(* IEC 61131-3 sources: volt/packages/volt-lsp-iec/test-corpus/bakon-nano/Device/Plc Logic/Application/POUs/MachineControl, 14 files *)

(* ---- InputControl.pou ---- *)
PROGRAM InputControl
VAR
	bStartPressed		: BOOL;
	tonDelayStartButton : TON;
END_VAR
%LANGUAGE ST
(*TODO: IO Direct aan Station IO Hangen*)
//The quick brown fox jumps over the lazy dog

(*Data from IO *)
//Digital
g_byInputs_Module_00			:= %IB8;
g_byInputs_Module_01			:= %IB9;
//Analog
g_wInputs_Module_00				:= %IW5;
g_wInputs_Module_01				:= %IW6;

(*first  module *)
g_bDI_ES_DirectOK				:= g_byInputs_Module_00.0;
g_bDI_CircuitBreaker_i700		:= g_byInputs_Module_00.1;
g_bDI_CircuitBreaker_Ultrasonic	:= g_byInputs_Module_00.2;
g_bDI_PressureSwitchOK			:= g_byInputs_Module_00.3;
bStartPressed					:= g_byInputs_Module_00.4 OR (bStartPressed AND NOT tonDelayStartButton.q);
g_bDI_LightCurtainOK			:= g_byInputs_Module_00.5;
g_bDI_MachineInSafePosition		:= g_byInputs_Module_00.6;
g_bDI_TableCheck				:= g_byInputs_Module_00.7;

(*second module *)
g_bDI_Servo_Power_OK			:= g_byInputs_Module_01.0;
g_bDI_CleaningContainerUp		:= g_byInputs_Module_01.1;	//Spare
g_bDI_CleaningContainerDown		:= g_byInputs_Module_01.2;	//Spare
g_bDI_UltraSonic_Error			:= g_byInputs_Module_01.3;
g_bDI_UltraSonic_ErrorCode_1	:= g_byInputs_Module_01.4;
g_bDI_UltraSonic_ErrorCode_2	:= g_byInputs_Module_01.5;
g_bDI_Spare16					:= g_byInputs_Module_01.6;
g_bDI_Spare17					:= g_byInputs_Module_01.7;

tonDelayStartButton(IN:=bStartPressed, PT:=T#500MS);
g_bDI_StartButton := tonDelayStartButton.Q;

(*fifth module *)
g_iAI_UltrasonicPower			:= TO_INT(TO_REAL(g_wInputs_Module_00)/16384);
g_iAI_Spare_01					:= TO_INT(TO_REAL(g_wInputs_Module_01)/16384);

END_PROGRAM

(* ---- MACH_AUT_Automatic.pou ---- *)
PROGRAM MACH_AUT_Automatic
VAR
	tWatchDogTimer					: TON;
	tStepTimer						: TOF;
	bwait                  			: BOOL;
	bPulseStepCounter      			: BOOL;
	bHoldPointOnReq        			: BOOL;
	bHoldPointOnErr3       			: BOOL;
	bStopPointAutomatic    			: BOOL;

	bOnePiece						: BOOL;
	bStartButtonPressed				: BOOL;
	nOldProductType					: INT;
	nOldNumberRoundParts			: INT;
	nDebugLastStep					: INT;
	bStartedOnce						: BOOL := FALSE;
	rt_PressStartToInit: R_TRIG;
	tofRecipeLoad					: TOF;
	bStartPressedWhileLoadeing	: BOOL := FALSE;
	sOldRecipeName					: STRING;
	tMachineInSafePosition			: TOF;
	bFirstTimeWaitForExec: BOOL;
	nScanCount : INT;
	bStartPressedWhileError : BOOL;
END_VAR
%LANGUAGE ST
(*************************************************************************
 *
 * Application name			: Snijmachine
 * Module name				: MACH_AUT_automatic
 * Version number module	: 1.00
 *
 *
 *                  Copyright (c) Bakon 2009
 *                  Goes, The Netherlands
 *
 *
 * All rights are reserved. Reproduction in whole or in part is prohibited
 * without the written consent of the copyright owner.
 *
 *************************************************************************)

(*************************************************************************
 * HISTORY
 *************************************************************************
 * Update  :
 * Author  :
 * Changes :
 *************************************************************************)

(****************************************************************************************************************************)
bHoldPointOnReq		:= FALSE;
bHoldPointOnErr3		:= FALSE;
bStopPointAutomatic		:= FALSE;

g_sMACH.aut.bActAutomatic     := g_sMACH.MCL.bActAutomatic;

(* Force C_NOT_ACTIVE state *)
IF     NOT g_sMACH.aut.bActAutomatic
THEN
		IF g_sMACH.aut.nStepCounter <> C_NOT_ACTIVE THEN
			nDebugLastStep := g_sMACH.aut.nStepCounter;
		END_IF
		g_sMACH.aut.nStepCounter := C_NOT_ACTIVE;
END_IF;

IF         g_sMACH.aut.nStepCounter <> C_NOT_ACTIVE
THEN
   (* -------------------------------------------------------------------------
    * Prestep Code
    * ------------------------------------------------------------------------- *)
	tofRecipeLoad(IN:=g_HMI_sRecipeName <> sOldRecipeName, PT:=T#3s);
	sOldRecipeName := g_HMI_sRecipeName;
	bStartPressedWhileLoadeing := bStartPressedWhileLoadeing OR (tofRecipeLoad.Q AND g_bDI_StartButton);

	IF NOT gMachConfig.bCleaningUnit THEN		// Voor de veiligheid...
		g_bCleanRequest := FALSE;
	END_IF

END_IF

(* Product not finished reset when new recipe or when in Testmode *)
IF		g_HMI_RCP_Parameters.nProductType <> nOldProductType
	OR	g_HMI_RCP_Parameters.nPartsRound <> nOldNumberRoundParts
	OR	g_HMI_MachCommand.bTestMode
	OR 	g_HMI_MachCommand.bScanMode
	OR	g_sMACH.ERR.bCalcVerError
	OR	g_sMACH.ERR.bCalcHorError
	OR	g_sMACH.ERR.bCalcDia1Error
	OR	g_sMACH.ERR.bCalcDia2Error
	OR	g_sMACH.ERR.bErrorPosNotPossible
	OR	g_sMACH.ERR.bPieceTooLarge
	OR	g_sMACH.ERR.bTrayTooSmall
THEN
	g_bProductNotFinished := FALSE;
END_IF
nOldProductType := g_HMI_RCP_Parameters.nProductType;
nOldNumberRoundParts := g_HMI_RCP_Parameters.nPartsRound;

(* Offdelay g_bDI_MachineInSafePosition tbv veilig starten cyclus*)
tMachineInSafePosition(IN := g_bDI_MachineInSafePosition, PT := t#800ms);

(* detect change of state *)
bPulseStepCounter     := g_sMACH.aut.nStepCounter <> g_sMACH.aut.nOldStepCounter;
g_sMACH.aut.nOldStepCounter := g_sMACH.aut.nStepCounter;

(* Steptimer *)
tStepTimer (IN:=bPulseStepCounter, PT:= REAL_TO_TIME(g_sMACH.AUT.rStepTime));
bWait := tStepTimer.Q;

(* Watchdogtimer *)
tWatchdogTimer(	IN:=		NOT	bPulseStepCounter
							AND 		g_sMACH.AUT.bActAutomatic
							AND NOT 	g_sMACH.AUT.bAutomatichold
							AND NOT 	g_HMI_MachCommand.CMD.bResetErrorPulse
							AND 		g_sMACH.AUT.rWatchdogTime<> 0,
					PT:= 	REAL_TO_TIME(g_sMACH.AUT.rWatchdogTime));
g_sMACH.AUT.bAlmError := tWatchdogTimer.Q;

(* Melding op scherm om startknop in te drukken *)
rt_PressStartToInit(CLK := (g_sMACH.Aut.nStepCounter = C_INITIAL));
IF	rt_PressStartToInit.Q THEN
	g_sMACH.ERR.bPressStartToInit	:= TRUE;
END_IF
IF		g_bSUB_InitStart
	OR	(g_sMACH.Aut.nStepCounter = C_NOT_ACTIVE)
THEN
	g_sMACH.ERR.bPressStartToInit	:= FALSE;
END_IF
g_sMACH.ERR.bPressStartToCut	:= g_sMACH.Aut.nStepCounter = C_WAIT_EXEC;

CASE g_sMACH.Aut.nStepCounter OF
	(* --------------------------------------------------------------------------
	 * S-1  C_NOT_ACTIVE
	 *      OnEntry: Ready  := FALSE
	 *      OnEntry: Busy   := FALSE
	 *      OnEntry: Hold   := FALSE
	 *      OnEntry: Reset all non-stored commands
	 * T000 Activate signal
	 * -------------------------------------------------------------------------- *)
	C_NOT_ACTIVE:

		(* On Entry *)
		IF	bPulseStepCounter
		THEN
			g_sMACH.AUT.rWatchdogTime  			:= 0;
			g_sMACH.AUT.rStepTime				:= 0;

			g_sMACH.AUT.bAutomaticReady			:= FALSE;
			g_sMACH.AUT.bAutomaticBusy			:= FALSE;
			g_sMACH.AUT.bAutomaticHold			:= FALSE;
			g_sMACH.AUT.bAutomaticStop			:= FALSE;
			g_sMACH.AUT.bProcessBusy			:= FALSE;
			g_sMACH.AUT.bProcessReady			:= FALSE;
			g_sMACH.AUT.bAutomaticWaitingForTrig	:= FALSE;

			g_bCalculationStart					:= FALSE;
			g_bSUB_InitStart					:= FALSE;
			g_bSUB_CleanKnifeStart				:= FALSE;

			g_bCMD_US_Start1					:= FALSE;

			ModusRV.bEnable					:= FALSE;
			ModusRV.bStartXYA					:= FALSE;
			ModusRV.bStartZ						:= FALSE;

			g_sHMI_Mach_UnitStatus.bProcessAgain	:= FALSE;
			bStartButtonPressed							:= FALSE;

			g_bSaveMachPar								:= bStartedOnce;

			g_HMI_MachCommand.CMD.bDeny			:= FALSE;
			g_HMI_MachCommand.CMD.bConfirm		:= FALSE;

			bStartPressedWhileLoadeing := FALSE;
			g_sMACH.ERR.bMessagePosNotPossible := FALSE;

			g_HMI_MachCommand.CMD.bCleanKnifeRequest	:= FALSE;
			g_sHMI_Mach_UnitStatus.bPopupRemoveProduct := FALSE;
		END_IF

		(* Continuous actions *)
		IF NOT g_HMI_MachCommand.bScanMode THEN
			nScanCount := 0;
		END_IF

		(* Transitions *)
		IF	g_sMACH.aut.bActAutomatic
		THEN
			g_sMACH.aut.nStepCounter         := C_INITIAL;
			bStartedOnce := TRUE;
		END_IF;

	(* --------------------------------------------------------------------------
	 * S000 Sub init before starting auto cycle
	 * T995 C_WAIT_EXEC, Pre init done
	 * -------------------------------------------------------------------------- *)
	C_INITIAL:

	      (* On Entry *)
	      IF	bPulseStepCounter
		THEN
			g_sMACH.AUT.rWatchdogTime  			:= 0;
			g_sMACH.AUT.rStepTime				:= 0;
			MACH_SUB_Initialise.I_rX_InfeedPosition		:= g_HMI_MCH_Parameters.rInfeedPosition_X;
			IF 		g_HMI_MachCommand.bTestMode
				OR 	g_HMI_MachCommand.bScanMode
			THEN
				MACH_SUB_Initialise.I_rY_InfeedPosition		:= g_HMI_MCH_Parameters.rInfeedPosition_Y + 30;
			ELSE
				MACH_SUB_Initialise.I_rY_InfeedPosition		:= g_HMI_MCH_Parameters.rInfeedPosition_Y;
			END_IF
			MACH_SUB_Initialise.I_rY_InfeedPrePosition	:= g_HMI_MCH_Parameters.rInfeedPosition_Y + 30;
		END_IF;

		(* Continuous actions *)
		IF	g_bDI_StartButton OR g_HMI_MachCommand.bScanMode
		THEN
			g_bSUB_InitStart							:= TRUE;
		END_IF

		(* Transitions *)
		IF		g_bSUB_InitDone
		THEN
				g_bSUB_InitStart				:= FALSE;
				g_sMACH.aut.nStepCounter	:= C_WAIT_EXEC;
				bStartPressedWhileLoadeing := FALSE;
		END_IF;

	(* --------------------------------------------------------------------------
	 * S995 C_WAIT_EXEC
	 *      AutomaticWaitingForTrig := NOT AutomaticStop
	 * T996 C_INITIALISE
	 *              Execution Trigger
	 *      AND NOT Hold On Request
	 *      AND NOT Hold On Error Category 3
	 *      AND NOT Stop end of cycle selected
	 *      AND NOT Stop at error category 2
	 * T997 C_STOPPED
	 *         "Stop end of cycle" selected
	 *      OR "Stop on error category 2"
	 * -------------------------------------------------------------------------- *)
	C_WAIT_EXEC:

	      (* Actions on state entry *)
		IF	bPulseStepCounter
		THEN
			g_sMACH.AUT.rWatchdogTime  			:= 0;
			g_sMACH.AUT.rStepTime				:= 0;
			g_sMACH.ERR.bMessagePosNotPossible := FALSE;
			g_sMACH.AUT.rWatchdogTime  			:= 0;
			IF	g_HMI_MachCommand.bScanMode AND NOT bFirstTimeWaitForExec THEN
				g_sMACH.AUT.rStepTime			:= 2000;
			ELSE
				g_sMACH.AUT.rStepTime				:= 0;
			END_IF
			IF g_sMACH.ERR.bCrashDetected THEN
				g_bProductNotFinished	:= FALSE;
				g_sHMI_Mach_UnitStatus.bPopupRemoveProduct	:= TRUE;	// Popup
			END_IF
			bStartPressedWhileError := FALSE;
		END_IF

		bStartPressedWhileError := bStartPressedWhileError OR (g_sMACH.ERR.bCrashDetected AND g_bDI_StartButton);

		(* Continuous actions *)
		bHoldPointOnReq     := TRUE;
		bHoldPointOnErr3    := TRUE;
		bStopPointAutomatic := TRUE;
		IF	g_HMI_MachCommand.CMD.bConfirm THEN
			g_sHMI_Mach_UnitStatus.bPopupRemoveProduct	:= FALSE;	// Popup
			g_HMI_MachCommand.CMD.bConfirm	:= FALSE;
			g_sMACH.ERR.bCrashDetected	:= FALSE;
		END_IF

		(* Transitions *)
		IF				g_sMACH.MCL.bStopEndOfCycle
				OR		g_sMACH.MCL.bStopOnErrorCat2
				OR 		(g_HMI_MachCommand.bScanMode AND nScanCount >= 10)
		THEN
			g_sMACH.aut.nStepCounter     		:= C_STOPPED;
			IF g_HMI_MachCommand.bScanMode THEN
				g_sHMI_Mach_UnitStatus.bScanFinished := TRUE;
				g_bScanDataPending := TRUE;
			END_IF
		ELSIF	((g_bDI_StartButton
			AND tMachineInSafePosition.Q)
			OR g_HMI_MachCommand.bTestMode
			OR	(g_HMI_MachCommand.bScanMode
			AND NOT bwait AND nScanCount < 10)
			OR (bStartPressedWhileLoadeing
			AND tMachineInSafePosition.Q)
			OR bStartPressedWhileError)
			AND g_bDI_LightCurtainOK
			AND NOT tofRecipeLoad.Q
			AND NOT g_sMACH.ERR.bCrashDetected
		THEN
			g_uControl_X_Axis.bEnableDrive		:= TRUE;
			g_uControl_Y_Axis.bEnableDrive		:= TRUE;
			g_uControl_Front_Axis.bEnableDrive	:= TRUE;
			g_uControl_Rear_Axis.bEnableDrive	:= TRUE;
			g_uControl_Z_Axis.bEnableDrive		:= TRUE;
			g_uControl_R_Axis.bEnableDrive		:= TRUE;

			bStartButtonPressed 				:= FALSE;
			bStartPressedWhileLoadeing	:= FALSE;
			g_sMACH.aut.nStepCounter		:= C_INITIALISE;
		END_IF

	(* --------------------------------------------------------------------------
	 * S996 C_INITIALISE
	 *      OnEntry: bProcessBusy  := TRUE
	 *      OnEntry: ProcessReady := FALSE
	 * T005 Always
	 * -------------------------------------------------------------------------- *)
	C_INITIALISE:

	      (* On entry *)
		IF	bPulseStepCounter
		THEN
			g_sMACH.aut.bProcessReady		:= FALSE;
			g_sMACH.aut.bProcessBusy		:= TRUE;
			g_sMACH.AUT.rWatchdogTime  		:= 10 * 1000;
			g_sMACH.AUT.rStepTime			:= 0;
	      END_IF

		(* Continuous actions *)
		IF g_sMACH.AUT.bAlmError THEN
			IF NOT g_uStatus_X_Axis.bDriveEnabled
				OR NOT g_uStatus_Y_Axis.bDriveEnabled
				OR NOT g_uStatus_Front_Axis.bDriveEnabled
				OR NOT g_uStatus_Rear_Axis.bDriveEnabled
			THEN
				g_sMACH.ERR.bXYNotEnabled := TRUE;
			END_IF
			IF NOT g_uStatus_Z_Axis.bDriveEnabled THEN
				g_sMACH.ERR.bZNotEnabled := TRUE;
			END_IF
			IF NOT g_uStatus_R_Axis.bDriveEnabled THEN
				g_sMACH.ERR.bRNotEnabled := TRUE;
			END_IF
		END_IF
		IF	g_HMI_MachCommand.CMD.bConfirm THEN
			g_sHMI_Mach_UnitStatus.bPopupRemoveProduct	:= FALSE;	// Popup
			g_HMI_MachCommand.CMD.bConfirm	:= FALSE;
			g_sMACH.ERR.bCrashDetected	:= FALSE;
		END_IF

		(* Transitions *)
		IF		g_uStatus_Z_Axis.bDriveEnabled
			AND	g_uStatus_R_Axis.bDriveEnabled
			AND	g_uStatus_X_Axis.bDriveEnabled
			AND	g_uStatus_Y_Axis.bDriveEnabled
			AND	g_uStatus_Rear_Axis.bDriveEnabled
			AND	g_uStatus_Front_Axis.bDriveEnabled
			AND NOT g_sMACH.ERR.bCrashDetected
		THEN
			g_sMACH.aut.nStepCounter	:= 010;
		END_IF

	(*--------------------------------------------------------------------------
	 * S010 Enable Modus RondVierkant
	 *		 Check if product has been cut completely
	 * T015 Always
	 * -------------------------------------------------------------------------- *)
	010:

	      (* On entry *)
		IF	bPulseStepCounter
		THEN
			g_sMACH.AUT.rWatchdogTime  				:= 0;
			g_sMACH.AUT.rStepTime					:= 0;
			ModusRV.bEnable 							:= TRUE;
			IF g_bProductNotFinished AND NOT g_HMI_MachCommand.bTestMode AND NOT g_HMI_MachCommand.bScanMode
			THEN
				g_sHMI_Mach_UnitStatus.bProcessAgain	:= TRUE;	(* Open popup in screen *)
			END_IF
		END_IF

		(* Continuous actions *)

		(* Transitions *)
		IF			(g_bProductNotFinished AND g_HMI_MachCommand.CMD.bDeny)
			OR		g_HMI_MachCommand.bTestMode
			OR 		g_HMI_MachCommand.bScanMode
			OR	NOT	g_bProductNotFinished
		THEN
			g_sHMI_Mach_UnitStatus.bProcessAgain	:= FALSE;	(* Popup in screen *)
			g_HMI_MachCommand.CMD.bDeny			:= FALSE;
			g_HMI_MachCommand.CMD.bConfirm		:= FALSE;
			g_sMACH.aut.nStepCounter	:= 015;
		ELSIF	(g_bProductNotFinished AND g_HMI_MachCommand.CMD.bConfirm)
		THEN
			g_sHMI_Mach_UnitStatus.bProcessAgain	:= FALSE;	(* Popup in screen *)
			g_HMI_MachCommand.CMD.bDeny			:= FALSE;
			g_HMI_MachCommand.CMD.bConfirm		:= FALSE;
			g_sMACH.aut.nStepCounter	:= 020;
		END_IF

	(*--------------------------------------------------------------------------
	 * S015 Calculate cutting positions
	 * T020 Calculations done
	 * -------------------------------------------------------------------------- *)
	015:

	      (* On entry *)
		IF	bPulseStepCounter
		THEN
			g_sMACH.AUT.rWatchdogTime  				:= 0;
			g_sMACH.AUT.rStepTime					:= 0;
			g_bCalculationStart							:= TRUE;

		END_IF

		(* Continuous actions *)
		bOnePiece	:= 		g_HMI_RCP_Parameters.rSizeTrimRight = 0 												(* No cuts when one piece and no trims *)
					AND	g_HMI_RCP_Parameters.rSizeTrimLeft = 0
					AND	g_HMI_RCP_Parameters.rSizeTrimRear = 0
					AND	g_HMI_RCP_Parameters.rSizeTrimFront = 0
					AND	g_HMI_RCP_Parameters.nPartsX = 1
					AND	g_HMI_RCP_Parameters.nPartsY = 1;

		(* Transitions *)
		IF			g_bCalculationDone
		THEN
			g_bCalculationStart				:= FALSE;
			g_sMACH.aut.nStepCounter		:= 020;
		END_IF

	(*--------------------------------------------------------------------------
	 * S020 Start cutting
	 * T025 Always
	 * -------------------------------------------------------------------------- *)
	020:

	      (* On entry *)
		IF	bPulseStepCounter
		THEN
			g_sMACH.AUT.rWatchdogTime  				:= 0;
			g_sMACH.AUT.rStepTime					:= 0;
			IF	NOT bOnePiece
			THEN
				ModusRV.bStartXYA	:= TRUE;
				ModusRV.bStartZ		:= TRUE;
				g_bProductNotFinished	:= TRUE;
				g_bCMD_US_Start1	:= TRUE;
			END_IF
		END_IF

		(* Continuous actions *)

		(* Transitions *)
		IF	TRUE
		THEN
			g_sMACH.aut.nStepCounter	:= 025;
		END_IF

	(*--------------------------------------------------------------------------
	 * S025 Wait for cutting ready
	 * T030 Cutting ready
	 * -------------------------------------------------------------------------- *)
	025:

	    (* On entry *)
		IF	bPulseStepCounter
		THEN
			g_sMACH.AUT.rWatchdogTime  				:= 0;
			g_sMACH.AUT.rStepTime					:= 0;
		END_IF

		(* Continuous actions *)

		(* Transitions *)
		IF		ModusRV.bLastCutReadyZOutOfProduct
			OR	ModusRV.bReady									(* @TODO, tekst bijzetten waarom, vermoedelijk voor als een product geen enkele keer gesneden moet worden *)
		THEN
			ModusRV.bStartXYA		:= FALSE;
			ModusRV.bStartZ			:= FALSE;
			g_bProductNotFinished	:= FALSE;
			g_sHMI_CountersInfinite.dnProductCountTotal	:= g_sHMI_CountersInfinite.dnProductCountTotal + 1;
			g_sHMI_CountersDay.dnProductCountTotal	:= g_sHMI_CountersDay.dnProductCountTotal + 1;
			g_bCMD_US_Start1	:= FALSE;

			IF NOT g_HMI_MachCommand.bScanMode AND NOT g_sMACH.ERR.bCrashDetected THEN
				CASE g_HMI_RCP_Parameters.nProductType OF
						Prod_Slab_Rectangle_1x1, Prod_Slab_Rectangle_1x1_Clamp:	(* ProductType = 0 = Slab Square *)
							g_sHMI_CountersInfinite.dnProductCountSlabSquare	:= 	g_sHMI_CountersInfinite.dnProductCountSlabSquare	+1;
							g_sHMI_CountersDay.dnProductCountSlabSquare		:= 	g_sHMI_CountersDay.dnProductCountSlabSquare	+1;
						Prod_Slab_Triangle_1x1:	(* ProductType = 1 = Slab triangle *)
							g_sHMI_CountersInfinite.dnProductCountSlabTriangle	:= 	g_sHMI_CountersInfinite.dnProductCountSlabTriangle	+1;
							g_sHMI_CountersDay.dnProductCountSlabTriangle	:= 	g_sHMI_CountersDay.dnProductCountSlabTriangle	+1;
						Prod_Slab_Diagonal_1x1:	(* ProductType = 2 = Slab diagonal *)
							g_sHMI_CountersInfinite.dnProductCountSlabDiagonal	:= 	g_sHMI_CountersInfinite.dnProductCountSlabDiagonal	+1;
							g_sHMI_CountersDay.dnProductCountSlabDiagonal		:= 	g_sHMI_CountersDay.dnProductCountSlabDiagonal	+1;
						Prod_Round_POC_2x1:	(* ProductType = 4 = Round Cake *)
							g_sHMI_CountersInfinite.dnProductCountRound		:= 	g_sHMI_CountersInfinite.dnProductCountRound + 2;
							g_sHMI_CountersDay.dnProductCountRound			:= 	g_sHMI_CountersDay.dnProductCountRound + 2;
						Prod_Tray_Rectangle_1x2, Prod_Tray_Rectangle_2x1:	(* ProductType = 4 = Tray Square Small *)
							g_sHMI_CountersInfinite.dnProductCountTraySmall		:= 	g_sHMI_CountersInfinite.dnProductCountTraySmall + 2;
							g_sHMI_CountersDay.dnProductCountTraySmall			:= 	g_sHMI_CountersDay.dnProductCountTraySmall + 2;
						Prod_Tray_Rectangle_1x1:	(* ProductType = 5 = Tray Square Large *)
							g_sHMI_CountersInfinite.dnProductCountTrayLarge		:= 	g_sHMI_CountersInfinite.dnProductCountTrayLarge +1;
							g_sHMI_CountersDay.dnProductCountTrayLarge			:= 	g_sHMI_CountersDay.dnProductCountTrayLarge +1;
						Prod_Tray_Rectangle_1x4:	(* ProductType =6 = Tray Square Triple *)
							g_sHMI_CountersInfinite.dnProductCountTrayTriple		:= 	g_sHMI_CountersInfinite.dnProductCountTrayTriple + 4;
							g_sHMI_CountersDay.dnProductCountTrayTriple			:= 	g_sHMI_CountersDay.dnProductCountTrayTriple + 4;
				END_CASE
			END_IF
			g_sMACH.aut.nStepCounter	:= 030;
		ELSIF	bOnepiece
		THEN
			ModusRV.bStartXYA			:= FALSE;
			ModusRV.bStartZ				:= FALSE;
			g_bProductNotFinished		:= FALSE;
			g_bCMD_US_Start1			:= FALSE;
			g_sMACH.aut.nStepCounter	:= 030;
		END_IF

	(*--------------------------------------------------------------------------
	 * S030 Wait for Modus ready
	 * T040 Cleaning
	 * T998 Modus ready
	 * -------------------------------------------------------------------------- *)
	030:

	      (* On entry *)
		IF	bPulseStepCounter
		THEN
			g_sMACH.AUT.rWatchdogTime  				:= 0;
			g_sMACH.AUT.rStepTime					:= 0;
		END_IF

		(* Continuous actions *)

		(* Transitions *)
		IF			ModusRV.bReady
				OR	bOnePiece
		THEN
(*			g_uControl_Front_Axis.bEnableDrive	:= FALSE;
			g_uControl_Rear_Axis.bEnableDrive	:= FALSE;
			g_uControl_Z_Axis.bEnableDrive		:= FALSE;
			g_uControl_R_Axis.bEnableDrive		:= FALSE;*)
			(*IF	g_bCleanRequest
			THEN
				g_bCleanRequest	:= FALSE;
				g_HMI_MachCommand.CMD.bCleanKnifeRequest	:= FALSE;
				g_sMACH.aut.nStepCounter	:= 40;
			ELSE *)
			g_uControl_X_Axis.bEnableDrive := FALSE;
			g_uControl_Y_Axis.bEnableDrive := FALSE;
			//g_HMI_MachCommand.CMD.bCleanKnifeRequest	:= FALSE;
			nScanCount := nScanCount + 1;
			g_sMACH.aut.nStepCounter	:= C_READY;
			//END_IF
		END_IF

	(*--------------------------------------------------------------------------
	 * S040 Cleaning
	 * T998 Modus ready
	 * -------------------------------------------------------------------------- *)
	040:

	      (* On entry *)
		IF	bPulseStepCounter
		THEN
			g_sMACH.AUT.rWatchdogTime  			:= 0;
			g_sMACH.AUT.rStepTime				:= 0;
			g_bSUB_CleanKnifeStart				:= TRUE;
		END_IF

		(* Continuous actions *)

		(* Transitions *)
		IF	g_bSUB_CleanKnifeDone
		THEN
(*			g_uControl_Front_Axis.bEnableDrive	:= FALSE;
			g_uControl_Rear_Axis.bEnableDrive	:= FALSE;
			g_uControl_Z_Axis.bEnableDrive		:= FALSE;
			g_uControl_R_Axis.bEnableDrive		:= FALSE;*)
			g_uControl_X_Axis.bEnableDrive	:= FALSE;
			g_uControl_Y_Axis.bEnableDrive	:= FALSE;
			g_bSUB_CleanKnifeStart			:= FALSE;
			g_sMACH.aut.nStepCounter		:= C_READY;
		END_IF

	(* --------------------------------------------------------------------------
	 * S998 C_READY
	 *      OnEntry: bProcessBusy  := FALSE
	 *      OnEntry: ProcessReady := TRUE
	 * T999 Always
	 * -------------------------------------------------------------------------- *)
	C_READY:

	      (* On Entry *)
		IF	bPulseStepCounter
		THEN
			g_sMACH.aut.bProcessBusy		:= FALSE;
			g_sMACH.aut.bProcessReady	:= TRUE;
			g_sMACH.aut.rWatchdogTime	:= 0;
		END_IF

		(* Continuous actions *)

		(* Transitions *)
		IF	TRUE
		THEN
			g_sMACH.AUT.rStepTime	:= 0;
			g_sMACH.aut.nStepCounter	:= C_LAST;
		END_IF

	(* --------------------------------------------------------------------------
	 * S997 C_STOPPED
	 *      OnEntry: AutomaticReady := TRUE
	 * T999     NOT "Stop end of cycle" selected
	 *      AND NOT "Stop on error category 2"
	 * -------------------------------------------------------------------------- *)
	C_STOPPED:

		(* On entry *)
		IF	bPulseStepCounter
		THEN
			g_sMACH.aut.rWatchdogTime     := 0;
		END_IF

		(* Continuous actions *)
		(*g_uControl_X_Axis.bEnableDrive	:=	FALSE; //g_uStatus_X_Axis.bAutomaticEnabled;
		g_uControl_Y_Axis.bEnableDrive	:=	FALSE; //g_uStatus_Y_Axis.bAutomaticEnabled;
		g_uControl_Front_Axis.bEnableDrive := FALSE; //g_uStatus_Front_Axis.bAutomaticEnabled;
		g_uControl_Rear_Axis.bEnableDrive := FALSE; //g_uStatus_Rear_Axis.bAutomaticEnabled;
		g_uControl_Z_Axis.bEnableDrive	:=	FALSE; //g_uStatus_Z_Axis.bAutomaticEnabled;
		g_uControl_R_Axis.bEnableDrive	:=	FALSE; //g_uStatus_R_Axis.bAutomaticEnabled;*)
		bStopPointAutomatic				:= TRUE;

		g_sMACH.Aut.bAutomaticReady    := TRUE;(*NOT (
													g_uStatus_X_Axis.bDriveEnabled
												OR	g_uStatus_Y_Axis.bDriveEnabled
												OR	g_uStatus_Front_Axis.bDriveEnabled
												OR	g_uStatus_Rear_Axis.bDriveEnabled
												OR	g_uStatus_Z_Axis.bDriveEnabled);*)

		(* Transitions *)
		IF		NOT g_sMACH.MCL.bStopEndOfCycle
			AND NOT g_sMACH.MCL.bStopOnErrorCat2
			AND NOT g_sHMI_Mach_UnitStatus.bScanFinished
		THEN
			g_sMACH.Aut.bAutomaticReady   := FALSE;
			g_sMACH.aut.nStepCounter      := C_LAST;
		END_IF

	(* --------------------------------------------------------------------------
	 * S999 C_LAST
	 * T000 Always
	 * -------------------------------------------------------------------------- *)
	C_LAST:

		(* On entry *)
		IF	bPulseStepCounter
		THEN
			g_sMACH.aut.rWatchdogTime     := 0;
		END_IF

		(* Continuous actions *)

		(* Transitions *)
		IF	TRUE THEN
			g_sMACH.aut.nStepCounter      := C_WAIT_EXEC;
		END_IF

	(* --------------------------------------------------------------------------
	 * Illegal state
	 * -------------------------------------------------------------------------- *)
ELSE
	g_sMACH.aut.rWatchdogTime     := 10;
END_CASE

IF      g_sMACH.Aut.nStepCounter <> C_NOT_ACTIVE
THEN
	(* --------------------------------------------------------------------------
	 * Poststep code
	 * -------------------------------------------------------------------------- *)
	g_sMACH.Aut.bAutomaticHold  :=	(	g_sMACH.MCL.bHoldOnRequest
									AND	bHoldPointOnReq)
									OR  (    g_sMACH.MCL.bHoldOnErrorCat3
									AND bHoldPointOnErr3);

	g_sMACH.Aut.bAutomaticStop  :=			bStopPointAutomatic
									AND	g_sMACH.MCL.bStopOnErrorCat2;

	g_sMACH.Aut.bAutomaticBusy  :=		NOT	g_sMACH.Aut.bAutomaticHold
										AND NOT	g_sMACH.Aut.bAutomaticStop;

	g_sMACH.Aut.bAutomaticWaitingForTrig :=        (g_sMACH.aut.nStepCounter = C_WAIT_EXEC)
												AND NOT g_sMACH.Aut.bAutomaticStop
												AND NOT g_sMACH.Aut.bAutomaticHold;
	g_sHMI_Mach_UnitStatus.nScanProgress := nScanCount;
END_IF

END_PROGRAM

(* ---- MACH_Call.pou ---- *)
PROGRAM MACH_Call
VAR
END_VAR
%LANGUAGE ST
(*************************************************************************
 *
 * Application name			: Snijmachine
 * Module name				: MACH_Call
 * Version number module	: 0.00
 *
 *                  Copyright (c) Bakon 2009
 *                  Goes, The Netherlands
 *
 *
 * All rights are reserved. Reproduction in whole or in part is prohibited
 * without the written consent of the copyright owner.
 *
 *************************************************************************)

(*************************************************************************
 * HISTORY
 *************************************************************************
 * Update  :
 * Author  :
 * Changes :
 *************************************************************************)

	(* -------------------------------------------------------------------------
	* Execution Control functions
	* ------------------------------------------------------------------------- *)
	MACH_HMI_Control();

	(* -------------------------------------------------------------------------
	* Execution Control functions
	* ------------------------------------------------------------------------- *)
	MACH_INI_Initialise();
(*    MACH_AUT_Automatic(); *)
	MACH_MAN_Manual();
	MACH_ERH_ErrorHandler();
	MACH_MCL_ModeControl();
	MACH_CLN_Cleaning();

	(* -------------------------------------------------------------------------
	* Drivers and calculations
	* ------------------------------------------------------------------------- *)
	MACH_DRV_DriverCall();
	Calc_Main();	(* Calculations *)

	(* -------------------------------------------------------------------------
	* Miscellaneous
	* ------------------------------------------------------------------------- *)
	MACH_MIS_Miscellaneous();
	MACH_ParameterHandler();
	RCP_RecipeHandler();
	HMI_ResetSignals();
	{warning 'Disabled for compatibility - SVE'}
	//g_Logger(directoryName := '/USBStorage/IPC/PLC/KC_Logs');

END_PROGRAM

(* ---- MACH_CLN_Cleaning.pou ---- *)
PROGRAM MACH_CLN_Cleaning
VAR
	bPulseStepCounter	: BOOL;
	bWait				: BOOL;
	tWatchDogTimer		: TON;
	tStepTimer			: TOF;
	rt_PressStartToInit	: R_TRIG;
END_VAR
%LANGUAGE ST
 (*************************************************************************
 *
 * Application name				: Snijmachine
 * Module name					: MACH_CLN_Cleaning
 * Version number module		: 0.00
 *
 *
 *						Copyright (c) Bakon 2009
 *						Goes, The Netherlands
 *
 *
 * All rights are reserved. Reproduction in whole or in part is prohibited
 * without the written consent of the copyright owner.
 *
 *************************************************************************)

(*************************************************************************
 * HISTORY
 *************************************************************************
 * Update  :
 * Author  :
 * Changes :
 *************************************************************************)

(* Force C_NOT_ACTIVE state *)
IF	NOT g_sMACH.MCL.bActCleaning
THEN
	g_sMACH.CLN.nStepCounter := C_NOT_ACTIVE;
END_IF;

IF		g_sMACH.CLN.nStepCounter <> C_NOT_ACTIVE
THEN
	(* -------------------------------------------------------------------------
	 * Prestep Code
	 * ------------------------------------------------------------------------- *)
				  ;
END_IF;

(* detect change of state *)
bPulseStepCounter	  := g_sMACH.CLN.nStepCounter <> g_sMACH.CLN.nOldStepCounter;
g_sMACH.CLN.nOldStepCounter := g_sMACH.CLN.nStepCounter;

(* Steptimer *)
tStepTimer (IN:= bPulseStepCounter, PT:= REAL_TO_TIME(g_sMACH.CLN.rStepTime));
bWait := tStepTimer.Q;

(* Watchdogtimer *)
tWatchDogTimer (IN:= 	NOT	bPulseStepCounter
					AND		g_sMACH.MCL.bActCleaning
					AND NOT	g_HMI_MachCommand.CMD.bResetErrorPulse
					AND		g_sMACH.CLN.rWatchdogTime <> 0,
				PT:= REAL_TO_TIME(g_sMACH.CLN.rWatchdogTime));
g_sMACH.CLN.bAlmError := tWatchDogTimer.Q;

(* Melding op scherm om startknop in te drukken *)
rt_PressStartToInit(CLK := (g_sMACH.CLN.nStepCounter = C_INITIAL));
IF	rt_PressStartToInit.Q THEN
	g_sMACH.ERR.bPressStartToCleanInit	:= TRUE;
END_IF
IF		g_bSUB_InitStart
	OR	(g_sMACH.CLN.nStepCounter = C_NOT_ACTIVE)
THEN
	g_sMACH.ERR.bPressStartToCleanInit	:= FALSE;
END_IF

CASE g_sMACH.CLN.nStepCounter OF
	(* --------------------------------------------------------------------------
	 * S-1  C_NOT_ACTIVE
	 *		OnEntry: Ready  := FALSE
	 *		OnEntry: Busy	:= FALSE
	 *		OnEntry: Reset all non-stored commands
	 * T000 Activate signal
	 * -------------------------------------------------------------------------- *)
	C_NOT_ACTIVE:

		(* On Entry *)
		IF		bPulseStepCounter
		THEN
				g_sMACH.CLN.rWatchdogTime					:= 0;
				g_sMACH.CLN.bCleaningReady					:= FALSE;
				g_sMACH.CLN.bCleaningBusy					:= FALSE;

				g_bSUB_InitStart							:= FALSE;

				g_HMI_MachCommand.CMD.bCleanKnifeRequest		:= FALSE;
				g_bSUB_CleanKnifeStart							:= FALSE;
				g_sHMI_Mach_UnitStatus.bKnifeCleaningBusy		:= FALSE;

				g_bCMD_US_Start1 							:= FALSE;
		END_IF

		(* Continuous actions *)

		(* Transitions *)
		IF		g_sMACH.MCL.bActCleaning
		THEN
				g_sMACH.CLN.nStepCounter			:= C_INITIAL;
		END_IF

	(* --------------------------------------------------------------------------
	 * S000 C_INITIAL
	 *		OnEntry: Ready := FALSE
	 *		OnEntry: Busy  := TRUE
	 *		Enable drives
	 * T001 Drives enabled
	 * -------------------------------------------------------------------------- *)
	C_INITIAL:

		(* On Entry *)
		IF		bPulseStepCounter
		THEN
				g_sMACH.CLN.rWatchdogTime					:= 0;
				g_sMACH.CLN.bCleaningReady					:= FALSE;
				g_sMACH.CLN.bCleaningBusy					:= TRUE;
		END_IF

		(* Continuous actions *)

		(* Transitions *)
		IF		g_sMACH.MCL.bStopEndOfCycle
		THEN
				g_sMACH.CLN.nStepCounter			:= C_READY;
		ELSIF			g_bDI_StartButton
				OR NOT	g_bDI_MachineInSafePosition
		THEN
				g_sMACH.CLN.nStepCounter			:= 005;
		END_IF

	(* --------------------------------------------------------------------------
	 * S005 Sub init before starting cleaning
	 * T010 Cleaning
	 * -------------------------------------------------------------------------- *)

	005:
		(* On Entry *)
	    IF	bPulseStepCounter
		THEN
			g_sMACH.CLN.rWatchdogTime  			:= 0;
			g_sMACH.CLN.rStepTime				:= 0;
			MACH_SUB_Initialise.I_rX_InfeedPosition		:= g_HMI_MCH_Parameters.rInfeedPosition_X;
			MACH_SUB_Initialise.I_rY_InfeedPosition		:= g_HMI_MCH_Parameters.rInfeedPosition_Y + 30;
			MACH_SUB_Initialise.I_rY_InfeedPrePosition	:= g_HMI_MCH_Parameters.rInfeedPosition_Y + 30;
		END_IF

		g_bSUB_InitStart						:= TRUE;

		(* Transitions *)
		IF	g_bSUB_InitDone
		THEN
			g_sMACH.CLN.nStepCounter			:= 010;
			g_bSUB_InitStart := FALSE;
		END_IF

	(* --------------------------------------------------------------------------
	 * S010 Enable drives
	 * T015 Drives enabled
	 * -------------------------------------------------------------------------- *)
	010:

		(* On Entry *)
		IF		 bPulseStepCounter
		THEN
				g_sMACH.CLN.rWatchdogTime			:= 10*1000;
				g_sMACH.CLN.rStepTime				:= 0;
				g_uControl_X_Axis.bEnableDrive		:= TRUE;
				g_uControl_Y_Axis.bEnableDrive		:= TRUE;
				g_uControl_Front_Axis.bEnableDrive	:= TRUE;
				g_uControl_Rear_Axis.bEnableDrive	:= TRUE;
				g_uControl_Z_Axis.bEnableDrive		:= TRUE;
				g_uControl_R_Axis.bEnableDrive		:= TRUE;
		END_IF

		(* Continuous actions *)
		IF g_sMACH.CLN.bAlmError THEN
			IF NOT g_uStatus_X_Axis.bDriveEnabled
				OR NOT g_uStatus_Y_Axis.bDriveEnabled
				OR NOT g_uStatus_Front_Axis.bDriveEnabled
				OR NOT g_uStatus_Rear_Axis.bDriveEnabled
			THEN
				g_sMACH.ERR.bXYNotEnabled := TRUE;
			END_IF
			IF NOT g_uStatus_Z_Axis.bDriveEnabled THEN
				g_sMACH.ERR.bZNotEnabled := TRUE;
			END_IF
			IF NOT g_uStatus_R_Axis.bDriveEnabled THEN
				g_sMACH.ERR.bRNotEnabled := TRUE;
			END_IF
		END_IF

		(* Transitions *)
		IF		g_uStatus_Z_Axis.bDriveEnabled// AND g_uStatus_Z_Axis.bAutomaticEnabled
			AND	g_uStatus_R_Axis.bDriveEnabled //AND g_uStatus_R_Axis.bAutomaticEnabled
			AND	g_uStatus_X_Axis.bDriveEnabled //AND g_uStatus_X_Axis.bAutomaticEnabled
			AND	g_uStatus_Y_Axis.bDriveEnabled //AND g_uStatus_Y_Axis.bAutomaticEnabled
			AND	g_uStatus_Rear_Axis.bDriveEnabled //AND g_uStatus_Rear_Axis.bAutomaticEnabled
			AND	g_uStatus_Front_Axis.bDriveEnabled //AND g_uStatus_Front_Axis.bAutomaticEnabled
		THEN
				  g_sMACH.CLN.nStepCounter				:= 15;
		END_IF

	(* --------------------------------------------------------------------------
	 * S015 Wait for request from HMI
	 * T020	Start cleaning
	 * T998 Never
	 * -------------------------------------------------------------------------- *)
	015:

		(* On Entry *)
		IF		 bPulseStepCounter
		THEN
				g_sMACH.CLN.rWatchdogTime			:= 0;
				g_sMACH.CLN.rStepTime				:= 0;
				//g_uControl_X_Axis.bEnableDrive		:= TRUE;
				//g_uControl_Y_Axis.bEnableDrive		:= TRUE;
				//g_uControl_Front_Axis.bEnableDrive	:= TRUE;
				//g_uControl_Rear_Axis.bEnableDrive	:= TRUE;
				//g_uControl_Z_Axis.bEnableDrive		:= TRUE;
				//g_uControl_R_Axis.bEnableDrive		:= TRUE;
				g_bCMD_US_Start1 						:= TRUE;
		END_IF

		(* Continuous actions *)
		IF		g_HMI_MachCommand.CMD.bCleanKnifeRequest
			OR	g_HMI_MachCommand.CMD.bTableToCleanPos
		THEN
			g_bSUB_CleanKnifeStart	:= TRUE;
		END_IF
		g_sHMI_Mach_UnitStatus.bKnifeCleaningBusy	:= g_bSUB_CleanKnifeStart AND NOT g_sMACH.SUBClean.bSubProcessBusy1;
		g_sHMI_Mach_UnitStatus.bCleaningTableBusy	:= g_bSUB_CleanKnifeStart AND g_sMACH.SUBClean.bSubProcessBusy1;

		IF	g_bSUB_CleanKnifeDone
		THEN
			g_HMI_MachCommand.CMD.bCleanKnifeRequest	:= FALSE;
			g_sHMI_Mach_UnitStatus.bCleaningTableBusy	:= FALSE;
			g_bSUB_CleanKnifeStart			:= FALSE;
		END_IF

		(* Transitions *)
		IF		NOT	g_bSUB_CleanKnifeStart
			AND	g_sMACH.MCL.bStopEndOfCycle
		THEN
				  g_sMACH.CLN.nStepCounter				:= C_READY;
		END_IF

	(* --------------------------------------------------------------------------
	 * S020	Start cleaning
	 * T15	Cleaning done
	 * -------------------------------------------------------------------------- *)
	020:

		(* On Entry *)
		IF		 bPulseStepCounter
		THEN
				g_sMACH.CLN.rWatchdogTime			:= 0;
				g_sMACH.CLN.rStepTime				:= 0;
				g_uControl_X_Axis.bEnableDrive		:= TRUE;
				g_uControl_Y_Axis.bEnableDrive		:= TRUE;
				g_uControl_Front_Axis.bEnableDrive	:= TRUE;
				g_uControl_Rear_Axis.bEnableDrive	:= TRUE;
				g_uControl_Z_Axis.bEnableDrive		:= TRUE;
				g_uControl_R_Axis.bEnableDrive		:= TRUE;
		END_IF

		IF		g_HMI_MachCommand.CMD.bCleanKnifeRequest
		THEN
			g_bSUB_CleanKnifeStart	:= TRUE;
		END_IF
		g_sHMI_Mach_UnitStatus.bKnifeCleaningBusy	:= g_bSUB_CleanKnifeStart;

		(* Transitions *)
		IF	g_bSUB_CleanKnifeDone
		THEN
			g_HMI_MachCommand.CMD.bCleanKnifeRequest:= FALSE;
			g_sHMI_Mach_UnitStatus.bKnifeCleaningBusy	:= FALSE;
			g_bSUB_CleanKnifeStart			:= FALSE;
			g_sMACH.CLN.nStepCounter		:= 15;
		END_IF

	(* --------------------------------------------------------------------------
	 * S998 C_READY
	 *		OnEntry: Ready		:= TRUE
	 *		OnEntry: Busy		 := FALSE
	 *		Always : Activate errorhandler
	 * T000 Never
	 * -------------------------------------------------------------------------- *)
	C_READY:

		(* On Entry *)
		IF			bPulseStepCounter
		THEN
					  g_sMACH.CLN.rWatchdogTime	:= 0;
					  g_sMACH.CLN.bCleaningReady	:= TRUE;
					  g_sMACH.CLN.bCleaningBusy		:= FALSE;
					g_bCMD_US_Start1 				:= FALSE;
		END_IF

		(* Continuous actions *)
		g_sMACH.CLN.bCleaningReady					:= TRUE;

		(* Transitions *)
		IF			FALSE
		THEN
					  g_sMACH.CLN.nStepCounter				:= C_INITIAL;
		END_IF

(* --------------------------------------------------------------------------
 * Illegal state
 * -------------------------------------------------------------------------- *)
ELSE
	(* Programming error: Illegal state *)
	g_sMACH.CLN.rWatchdogTime := 10;
END_CASE;

IF			g_sMACH.CLN.nStepCounter <> C_NOT_ACTIVE
THEN
	(* -------------------------------------------------------------------------
	 * Poststep Code
	 * ------------------------------------------------------------------------- *)
	;
END_IF

END_PROGRAM

(* ---- MACH_DRV_DriverCall.pou ---- *)
PROGRAM MACH_DRV_DriverCall (* call all cylinder drivers *)
VAR
	Ultrasonic1		: DRV_AGM_IO;
	tMainValve		: TOF;
	Cyl_Cleaning	: DRV_CYL1C2D_SafeEnd;
	bCylCleaningCylUpAllowed	: BOOL;
END_VAR
%LANGUAGE ST
(**********************************************************************************************************)
(*Lampen & Signalen*)
(**********************************************************************************************************)
(*Drv_Lights(
	I_bErrorLevel4:= IQ_sTWD_Data.ERH.bErrorCategory4,
	I_bErrorLevel32:= IQ_sTWD_Data.ERH.bErrorCategory3 OR IQ_sTWD_Data.ERH.bErrorCategory2,
	I_bInitialising:= IQ_sTWD_Data.MCL.bActInitialise,
	I_bWaitForAutomatic:= IQ_sTWD_Data.MCL.nStepCounter = 6,
	I_bAutomatic:= IQ_sTWD_Data.MCL.bActAutomatic,
	I_bESActive:= NOT IQ_sIO_DATA.bDI_SafetyOK,
	I_bFilling:= IQ_sIO_DATA.bDQ_ProductRequest,
	I_bMachineAtTemp:= IQ_sTWD_Data.sHeatingStatus.bTempInTarget OR (sRCP_Parameters.nEnableHeating = 0),
	I_sControl:= IQ_sTWD_Data.sLights,
	Q_bMachinestandby=> ,	Q_bDepositActive=> IQ_sIO_DATA.bDQ_DepositActive,
	Q_bMachineFault=> IQ_sIO_DATA.bDQ_MachineFaultActive,
	Q_bGreenLight=> IQ_sIO_DATA.bDQ_MachineStandby,	(*AC Dit is misschien niet helemaal logisch bedraad?....*)
	Q_bOrangeLight=>IQ_sIO_DATA.bDQ_SignalOrange ,
	Q_bRedLight=> IQ_sIO_DATA.bDQ_SignalRed);
*)

(***************************************************************************************************************************)

(**********************************************************************************************************)
(* Airvalve:  *)
(**********************************************************************************************************)
tMainValve(IN := (g_sMACH.aut.bActAutomatic AND g_bDI_StartButton) OR g_bDQ_Ultrasonic1, PT := REAL_TO_TIME(g_HMI_MCH_Parameters.rTimeSwitchOffAirvalve * 60 * 1000));	(* Input HMI in minutes! *)
g_bDQ_MainValve := tMainValve.Q;

(**********************************************************************************************************)
(* Ultrasonic AGM *)
(**********************************************************************************************************)
Ultrasonic1(
	I_bCMD_Enable		:= g_bDI_ES_DirectOK AND (g_HMI_MCH_Parameters.bUltrasonicEnable1 OR g_sMACH.MCL.bActManual),
	I_bCMD_Start		:= (g_bCMD_US_Start1 AND NOT g_HMI_MachCommand.bScanMode) AND (g_bUS_EnableRV OR g_bUS_EnableCleaning),
	I_bCMD_Test			:= g_bCMD_US_Test1 OR (g_bCMD_US_Start1 AND g_HMI_MachCommand.bScanMode),			(* Only manual command *)
	I_bCMD_Reset		:= (g_HMI_MCH_Parameters.bUltrasonicEnable1 AND g_HMI_MachCommand.CMD.bResetErrorPulse),
	Q_bStart_AGM		:= g_bDQ_Ultrasonic1,
	Q_bTest_AGM			:= g_bTestAGM1);

(**********************************************************************************************************)
(* Cylinder Cleaning water container *)
(**********************************************************************************************************)
IF	gMachConfig.bCleaningUnit
THEN
	g_sMACH.sCleaningContainerControl.bErrorReset := g_HMI_MachCommand.CMD.bResetErrorPulse;

	bCylCleaningCylUpAllowed :=	(g_uStatus_X_Axis.lrActPosition <= 3)// g_HMI_MCH_Parameters.rCleanXPosStart + 1)(*Veilig indien messen voor x positie staan!*)
							AND ((g_uStatus_X_Axis.eStateAxis = L_MC1P_AXIS_STATE.StandStill) OR (g_uStatus_X_Axis.eStateAxis = L_MC1P_AXIS_STATE.Disabled))
							//AND (g_uStatus_Y_Axis.lrActPosition >= g_HMI_MCH_Parameters.rCleanYPosStop - 1)
							//AND ((g_uStatus_Y_Axis.eStateAxis = L_MC1P_AXIS_STATE.StandStill) OR (g_uStatus_Y_Axis.eStateAxis = L_MC1P_AXIS_STATE.Disabled))
							//AND	(g_uStatus_R_Axis.lrActPosition > 89.0)
							//AND	(g_uStatus_R_Axis.lrActPosition < 91.0)
							AND ((g_uStatus_R_Axis.eStateAxis = L_MC1P_AXIS_STATE.StandStill) OR (g_uStatus_R_Axis.eStateAxis = L_MC1P_AXIS_STATE.Disabled));

	Cyl_Cleaning(
		I_bCylEndPos	:= g_bDI_CleaningContainerUp,
		I_bCylZeroPos	:= g_bDI_CleaningContainerDown,
		I_bSafeEndOK		:= bCylCleaningCylUpAllowed,
		I_sControl		:= g_sMACH.sCleaningContainerControl,
		I_rTimeOut		:= g_HMI_MCH_Parameters.rCleanContainerTimeOut,
		DRV_ERR_CylEndPos:= g_sMACH.ERR.bCleaningContainerEndPos,
		DRV_ERR_CylZeroPos:= g_sMACH.ERR.bCleaningContainerZeroPos,
		DRV_ERR_CylMultiple:= g_sMACH.ERR.bCleaningContainerEndZero,
		DRV_ERR_SafetyNOK	:= g_sMACH.ERR.bCleaningContainerNotSafeToMove,
		Q_bCylToEndPos	=> g_bDQ_CleaningContainerUp,
		Q_bCylToZeroPos	=> g_bDQ_CleaningContainerDown,
		Q_sStatus		=> g_sMACH.sCleaningContainerStatus);

ELSE
		g_sMACH.ERR.bCleaningContainerEndPos	:= FALSE;
		g_sMACH.ERR.bCleaningContainerZeroPos	:= FALSE;
		g_sMACH.ERR.bCleaningContainerEndZero	:= FALSE;
		g_sMACH.ERR.bCleaningContainerNotSafeToMove	:= FALSE;
END_IF

END_PROGRAM

(* ---- MACH_ERH_ErrorHandler.pou ---- *)
PROGRAM MACH_ERH_ErrorHandler
VAR
	bSkipFirstTrigger		: BOOL	:= TRUE;
	tBuzzerTimerErr1		:TON;
	tBuzzerTimerErr234	:TON;
	Blinker					:BLINK;
	TON_Pressure		:TON;
	rSizeOfKnife			: REAL;
	rCenterPointKnifeInverted: REAL;
	rLengthOfLineHor: REAL;
	rLengthOfLineVer: REAL;
	bPosXaxisOK		: BOOL;
	bPosYaxisOK		: BOOL;
	bscandatapending : BOOL;

	tonTimeoutHomingDown: TON;
END_VAR
%LANGUAGE ST
(*************************************************************************
 *
 * Application name			: Snijmachine
 * Module name				: MACH_ERH_ErrorHandler
 * Version number module	: 0.00
 *
 *
 *						Copyright (c) Bakon 2009
 *						Goes, The Netherlands
 *
 *
 * All rights are reserved. Reproduction in whole or in part is prohibited
 * without the written consent of the copyright owner.
 *
 *************************************************************************)

(*************************************************************************
 * HISTORY
 *************************************************************************
 * Update  :
 * Author  :
 * Changes :
 *************************************************************************)

(* initialise signals on g_bFirstCycle *)
IF			g_bFirstCycle
THEN
			g_sMACH.ERH.bErrorCategory1		 := FALSE;
			g_sMACH.ERH.bErrorCategory2		 := FALSE;
			g_sMACH.ERH.bErrorCategory3		 := FALSE;
			g_sMACH.ERH.bErrorCategory4		 := FALSE;
			g_sMACH.ERH.bError234Active		:= FALSE;
			g_sMACH.ERH.bSoundSignalOn	:= FALSE;
END_IF

(* Reset the NOT-self resetting errors *)
IF		g_HMI_MachCommand.CMD.bResetErrorPulse
	OR	g_bFirstCycle
THEN
	g_sMACH.ERR.bEmergencyCircuitNotOK					:= FALSE;
	g_sMACH.ERR.ModusRV_AccDeccZ						:= FALSE;
	g_sMACH.ERR.ModusRV_SpeedZToHigh					:= FALSE;
	g_sMACH.ERR.ModusRV_TargetPosInSWLimits				:= FALSE;
	g_sMACH.ERR.bPressure								:= FALSE;
	g_sMACH.ERR.bErrorComIOStation						:= FALSE;
	g_sMACH.ERR.bTrayTooSmall							:= FALSE;
	g_sMACH.ERR.bR_AxisPositionError					:= FALSE;
	g_sMACH.ERR.bUltrasonic1							:= FALSE;
	g_sMACH.ERR.bAGM1_CommFailure						:= FALSE;
	g_sMACH.ERR.bPieceTooLarge							:= FALSE;
	g_sMACH.ERR.bAxisFrontNotSet						:= FALSE;
	g_sMACH.ERR.bAxisRearNotSet							:= FALSE;
	g_sMACH.ERR.bAxisRNotSet							:= FALSE;
	g_sMACH.ERR.bWrongTable								:= FALSE;
	g_sMACH.ERR.bSlabTooSmall							:= FALSE;
	g_sMACH.ERR.bXYNotEnabled							:= FALSE;
	g_sMACH.ERR.bZNotEnabled							:= FALSE;
	g_sMACH.ERR.bRNotEnabled							:= FALSE;
	g_sMACH.ERR.bServoPowerNOK							:= FALSE;
	g_sMACH.ERR.bTableMovementNotAllowed				:= FALSE;
	g_sMACH.ERR.bRAxisMovementNotAllowed				:= FALSE;
	g_sMACH.ERR.bZAxisMovementNotAllowed				:= FALSE;
	g_smach.ERR.bZHomeSensorTimeout						:= FALSE;
	g_sMACH.ERR.bCrashDetectFault						:= FALSE;
	g_sMACH.ERR.bStackIsFull							:= FALSE;
	g_sMACH.ERR.bStackIsEmpty							:= FALSE;
	g_sMACH.ERR.bMarginsInOvershootCorrectionInvalid	:= FALSE;
	g_sMACH.ERR.bKnifeSettingsIncorrect					:= FALSE;
	g_sMACH.ERR.bIntersectionNotFound					:= FALSE;
	g_sMACH.ERR.bOvershootCorrectionImpossible			:= FALSE;
	g_sMACH.ERR.bOldOvershootCorrectionDiffers			:= FALSE;
	g_sMACH.ERR.bIndexOutOfBoundsWhileCopyingCuts		:= FALSE;
	g_sMACH.ERR.bRoundProductsOverlap					:= FALSE;
	g_sMACH.ERR.bCalcVerError							:= FALSE;
	g_sMACH.ERR.bCalcHorError							:= FALSE;
	g_sMACH.ERR.bCalcDia1Error							:= FALSE;
	g_sMACH.ERR.bCalcDia2Error							:= FALSE;
	g_sMACH.ERR.bXYA_K_WasNotZero						:= FALSE;

	bscandatapending 								:= g_bFirstCycle;
END_IF

bscandatapending := bscandatapending AND g_bScanDataPending;
(* NOT-self resetting errors *)
(* Set_your_not_self_resetting_errors_here *)
IF	 NOT g_bDI_ES_DirectOK
THEN
		g_sMACH.ERR.bEmergencyCircuitNotOK := TRUE;
END_IF
IF	ModusRondVierkant.Q_bErrorAccDeccZ
THEN
	g_sMACH.ERR.ModusRV_AccDeccZ	 := TRUE;
END_IF
IF ModusRondVierkant.Q_bErrorSpeedZToHigh
THEN
	g_sMACH.ERR.ModusRV_SpeedZToHigh := TRUE;
END_IF
IF ModusRondVierkant.Q_bErrorTargetPosInSWLimits
THEN
	g_sMACH.ERR.ModusRV_TargetPosInSWLimits := TRUE;
END_IF
TON_Pressure(IN:= (NOT g_bDI_PressureSwitchOK AND g_bDQ_MainValve AND g_bDI_ES_DirectOK), pt:=REAL_TO_TIME(g_HMI_MCH_Parameters.rTimeOutAirvalve * 1000));
IF  TON_Pressure.Q THEN
	g_sMACH.ERR.bPressure := TRUE;
END_IF;

IF NOT g_bDI_Servo_Power_OK THEN
	g_sMACH.ERR.bServoPowerNOK := TRUE;
END_IF

tonTimeoutHomingDown(IN:=g_uStatus_Z_Axis.bHomingBusy AND g_uStatus_Z_Axis.bLimitNeg, PT:=T#3S);
IF tonTimeoutHomingDown.Q THEN
	g_sMACH.ERR.bZHomeSensorTimeout := TRUE;
END_IF
(*TODO: Via ethercat bepalen*)
(*IF g_aCanNodeState[C_NodeRemoteIO].xPdoTimeOut OR g_aCanNodeState[C_NodeRemoteIO].iState <> CanSlave_Operational THEN
IF EPM_S130.
	g_sMACH.ERR.bErrorComIOStation:=TRUE;
END_IF*)

(* Cleaning error *)
bPosXaxisOK := 	(g_uStatus_X_Axis.eStateAxis = L_MC1P_AXIS_STATE.StandStill)
			OR 	(g_uStatus_X_Axis.eStateAxis = L_MC1P_AXIS_STATE.Stopping)
			OR 	(g_uStatus_X_Axis.eStateAxis = L_MC1P_AXIS_STATE.Disabled)
			OR	(g_uStatus_X_Axis.lrActPosition <= C_rXAxis_SafeCleaningPos AND (NOT g_bDI_CleaningContainerDown OR NOT gMachConfig.bCleaningUnit))
			OR	(g_uStatus_X_Axis.lrActPosition <= g_HMI_MCH_Parameters.rCleanXPosStart + 1 AND (g_bDI_CleaningContainerDown OR NOT gMachConfig.bCleaningUnit));
bPosYaxisOK := 	(g_uStatus_Y_Axis.eStateAxis = L_MC1P_AXIS_STATE.StandStill)
			OR	(g_uStatus_Y_Axis.eStateAxis = L_MC1P_AXIS_STATE.Stopping)
			OR	(g_uStatus_Y_Axis.eStateAxis = L_MC1P_AXIS_STATE.Disabled)
			OR	(g_uStatus_X_Axis.lrActPosition < C_rXAxis_SafeCleaningPos AND (NOT g_bDI_CleaningContainerDown OR NOT gMachConfig.bCleaningUnit))		// X-as positie moet altijd OK zijn, ook bij de Y beweging
			OR	(g_uStatus_X_Axis.lrActPosition < g_HMI_MCH_Parameters.rCleanXPosStart + 1 AND (g_bDI_CleaningContainerDown OR NOT gMachConfig.bCleaningUnit));	// X-as positie moet altijd OK zijn, ook bij de Y beweging

IF		//NOT	g_sMACH.MCL.bActInitialise
			(NOT bPosXaxisOK OR NOT bPosYaxisOK)
	AND		((g_uStatus_Z_Axis.lrActPosition > g_sCalculated.rBottomZPos) OR (NOT g_bDI_CleaningContainerDown AND gMachConfig.bCleaningUnit))
THEN
	g_sMACH.ERR.bTableMovementNotAllowed	:= TRUE;
END_IF

IF		(g_uStatus_Z_Axis.lrActPosition > g_sCalculated.rBottomZPos)
	AND (g_uStatus_R_Axis.eStateAxis <> L_MC1P_AXIS_STATE.StandStill)
	AND (g_uStatus_R_Axis.eStateAxis <> L_MC1P_AXIS_STATE.Disabled)
	AND (g_uStatus_R_Axis.eStateAxis <> L_MC1P_AXIS_STATE.Stopping)
THEN
	g_sMACH.ERR.bRAxisMovementNotAllowed	:= TRUE;
END_IF

IF		(g_uStatus_Z_Axis.lrActPosition > g_sCalculated.rBottomZPos + 1)
	AND	g_uStatus_Z_Axis.bHomePositionAvailable
	AND (g_uStatus_Z_Axis.eStateAxis <> L_MC1P_AXIS_STATE.StandStill)
	AND (g_uStatus_Z_Axis.eStateAxis <> L_MC1P_AXIS_STATE.Disabled)
	AND (g_uStatus_Z_Axis.eStateAxis <> L_MC1P_AXIS_STATE.Stopping)
	AND	NOT g_uControl_Z_Axis.bManualJogNeg
	AND (g_uControl_Z_Axis.lrPosition <> 0 OR NOT g_uControl_Z_Axis.bPosABSPosition)
	AND ((g_uStatus_R_Axis.lrActPosition > 91.0) OR (g_uStatus_R_Axis.lrActPosition < 89.0) OR (g_uStatus_X_Axis.lrActPosition > g_HMI_MCH_Parameters.rCleanXPosStart + 1))
THEN
	g_sMACH.ERR.bZAxisMovementNotAllowed	:= TRUE;
END_IF

rSizeOfKnife				:= g_HMI_MCH_Parameters.rSizeOfKnife;
rCenterPointKnifeInverted	:= rSizeOfKnife/2;

(* Self resetting errors *)
(* Assign_your_self_resetting_errors_here (error := problem) *)
(* Check if machine parameters are not corrupted *)
g_sMACH.ERR.bZStrokeKnifeToBottomRound		:= (g_HMI_MCH_Parameters.rBottomZPosRound > C_LimitKnifeStrokeMax OR g_HMI_MCH_Parameters.rBottomZPosRound < C_LimitKnifeStrokeMin)
											AND (gProductOption.Prod_Round OR gProductOption.Prod_RoundQuatro);
g_sMACH.ERR.bZStrokeKnifeToBottomSlab		:= (g_HMI_MCH_Parameters.rBottomZPosSlab > C_LimitKnifeStrokeMax OR g_HMI_MCH_Parameters.rBottomZPosSlab < C_LimitKnifeStrokeMin)
											AND	(gProductOption.Prod_SlabDiagonal OR gProductOption.Prod_SlabDouble OR gProductOption.Prod_SlabSquare OR gProductOption.Prod_SlabSquareClamp OR gProductOption.Prod_SlabTriangle);
g_sMACH.ERR.bZStrokeKnifeToBottomTraySmall	:= (g_HMI_MCH_Parameters.rBottomZPosTraySmall > C_LimitKnifeStrokeMax OR g_HMI_MCH_Parameters.rBottomZPosTraySmall < C_LimitKnifeStrokeMin)
											AND (gProductOption.Prod_TraySquareSmall);
g_sMACH.ERR.bZStrokeKnifeToBottomTrayLarge	:= (g_HMI_MCH_Parameters.rBottomZPosTrayLarge > C_LimitKnifeStrokeMax OR g_HMI_MCH_Parameters.rBottomZPosTrayLarge < C_LimitKnifeStrokeMin)
											AND (gProductOption.Prod_TraySquareLarge);
g_sMACH.ERR.bZStrokeKnifeToBottomTrayDouble	:= (g_HMI_MCH_Parameters.rBottomZPosTrayDouble > C_LimitKnifeStrokeMax OR g_HMI_MCH_Parameters.rBottomZPosTrayDouble < C_LimitKnifeStrokeMin)		(* V07.01 *)
											AND (gProductOption.Prod_TraySquareDouble);
g_sMACH.ERR.bRoundCakeTooLarge				:=		g_HMI_RCP_Parameters.rDiameterRound  >= (g_HMI_MCH_Parameters.rMidPosRoundCake1_X - g_HMI_MCH_Parameters.rMidPosRoundCake2_X)
												AND g_HMI_RCP_Parameters.nProductType = Prod_Round_POC_2x1
												AND (g_HMI_RCP_Parameters.nPartsRound <> 0) AND (g_HMI_RCP_Parameters.nPartsRoundRight <> 0);		(* If only one cake is cut, then no error is created *)
g_sMACH.ERR.bRoundCakeTooLarge				:=	g_sMACH.ERR.bRoundCakeTooLarge OR
													g_HMI_RCP_Parameters.rDiameterRound  >= (g_HMI_MCH_Parameters.rMidPosRoundCake13_X - g_HMI_MCH_Parameters.rMidPosRoundCake24_X)
												OR g_HMI_RCP_Parameters.rDiameterRound  >= (g_HMI_MCH_Parameters.rMidPosRoundCake34_Y - g_HMI_MCH_Parameters.rMidPosRoundCake12_Y)
												AND	g_HMI_RCP_Parameters.nProductType = Prod_Round_POC_2x2;

rLengthOfLineHor := g_HMI_RCP_Parameters.rProdLength_InX - g_HMI_RCP_Parameters.rSizeTrimRight - g_HMI_RCP_Parameters.rSizeTrimLeft + (g_HMI_RCP_Parameters.nPartsX * g_HMI_RCP_Parameters.rShiftCompensation);
rLengthOfLineVer := g_HMI_RCP_Parameters.rProdLength_InY - g_HMI_RCP_Parameters.rSizeTrimFront - g_HMI_RCP_Parameters.rSizeTrimRear + (g_HMI_RCP_Parameters.nPartsY * g_HMI_RCP_Parameters.rShiftCompensation);
g_sMACH.ERR.bLengthExceededWithShiftComp	:=		(g_HMI_RCP_Parameters.nProductType = Prod_Slab_Rectangle_1x1)
														AND	(
																(rLengthOfLineHor > (SEL(gMachConfig.bXL,C_rMaxOvershootX,(C_rMaxOvershootX_XL) - g_HMI_MCH_Parameters.rStartPointSlab_X - g_HMI_RCP_Parameters.rSizeTrimRight)))
															OR	(rLengthOfLineVer > (SEL(gMachConfig.bXL,C_rMaxOvershootY,(C_rMaxOvershootY_XL) - g_HMI_MCH_Parameters.rStartPointSlab_Y - g_HMI_RCP_Parameters.rSizeTrimRear))));
g_sMACH.ERR.Z_AxisLimitNeg := g_uStatus_Z_Axis.bLimitNeg;		(* Standard V08.01*)
(* --------------------------------------------------------------------------
 * Assign errors of category 1 (Warnings)
 * -------------------------------------------------------------------------- *)
g_sMACH.ERR.dwCat1_Error.0 := g_sMACH.uINI.bAlmError;
g_sMACH.ERR.dwCat1_Error.1 := EtherCAT_Master.wState <> L_ETC.ETC_STATE_OPERATIONAL;//(g_aCanMasterState[0] <> CanMaster_Operational);
g_sMACH.ERR.dwCat1_Error.2 := g_sMACH.AUT.bAlmError;
g_sMACH.ERR.dwCat1_Error.3 := g_sMACH.MAN.bAlmError;
g_sMACH.ERR.dwCat1_Error.4 := g_sMACH.CLN.bAlmError;
g_sMACH.ERR.dwCat1_Error.5 := FALSE;
g_sMACH.ERR.dwCat1_Error.6 := g_sMACH.ERR.bErrorSetRef_Front_Axis;
g_sMACH.ERR.dwCat1_Error.7 := g_sMACH.ERR.bErrorSetRef_Rear_Axis;
g_sMACH.ERR.dwCat1_Error.8 := g_sMACH.ERR.bErrorSetRef_R_Axis;
g_sMACH.ERR.dwCat1_Error.9 := g_sMACH.ERR.bMaintenanceNecessary;
g_sMACH.ERR.dwCat1_Error.10 := g_sMACH.ERR.bAGM1_CommFailure;
g_sMACH.ERR.dwCat1_Error.11 := g_sMACH.ERR.bPressStartToInit;
g_sMACH.ERR.dwCat1_Error.12 := g_sMACH.ERR.bPressStartToCut AND NOT g_HMI_MachCommand.bScanMode;
g_sMACH.ERR.dwCat1_Error.13 := g_sMACH.ERR.bPressStartForManual;
g_sMACH.ERR.dwCat1_Error.14 := g_sMACH.ERR.bLengthExceededWithShiftComp;
g_sMACH.ERR.dwCat1_Error.15 := g_sMACH.ERR.Z_AxisLimitNeg;
g_sMACH.ERR.dwCat1_Error.16 := g_sMACH.ERR.bOvershootCorrectionImpossible AND g_HMI_MCH_Parameters.bSkipImpossiblePositions; //g_sMACH.ERR.bMessagePosNotPossible;
g_sMACH.ERR.dwCat1_Error.17 := g_sMACH.ERR.bPressStartToCleanInit;
g_sMACH.ERR.dwCat1_Error.18 := bscandatapending;
g_sMACH.ERR.dwCat1_Error.19 := g_sMACH.ERR.bCrashDetected;

(* --------------------------------------------------------------------------
 * Assign errors of category 2 (Stop at end of cycle)
 * -------------------------------------------------------------------------- *)
g_sMACH.ERR.dwCat2_Error.0 := FALSE;
g_sMACH.ERR.dwCat2_Error.1 := FALSE;
g_sMACH.ERR.dwCat2_Error.2 := FALSE;
g_sMACH.ERR.dwCat2_Error.3 := FALSE;
g_sMACH.ERR.dwCat2_Error.4 := FALSE;
g_sMACH.ERR.dwCat2_Error.5 := FALSE;
g_sMACH.ERR.dwCat2_Error.6 := FALSE;
g_sMACH.ERR.dwCat2_Error.7 := FALSE;
g_sMACH.ERR.dwCat2_Error.8 := FALSE;
g_sMACH.ERR.dwCat2_Error.9 := FALSE;
g_sMACH.ERR.dwCat2_Error.10 := FALSE;
g_sMACH.ERR.dwCat2_Error.11 := FALSE;
g_sMACH.ERR.dwCat2_Error.12 := FALSE;
g_sMACH.ERR.dwCat2_Error.13 := FALSE;
g_sMACH.ERR.dwCat2_Error.14 := FALSE;
g_sMACH.ERR.dwCat2_Error.15 := FALSE;

(* --------------------------------------------------------------------------
 * Assign errors of category 3 (Hold automatic)
 * -------------------------------------------------------------------------- *)
g_sMACH.ERR.dwCat3_Error.0 := FALSE;
g_sMACH.ERR.dwCat3_Error.1 := FALSE;
g_sMACH.ERR.dwCat3_Error.2 := FALSE;
g_sMACH.ERR.dwCat3_Error.3 := FALSE;
g_sMACH.ERR.dwCat3_Error.4 := FALSE;
g_sMACH.ERR.dwCat3_Error.5 := FALSE;
g_sMACH.ERR.dwCat3_Error.6 := FALSE;
g_sMACH.ERR.dwCat3_Error.7 := FALSE;
g_sMACH.ERR.dwCat3_Error.8 := FALSE;
g_sMACH.ERR.dwCat3_Error.9 := FALSE;
g_sMACH.ERR.dwCat3_Error.10 := FALSE;
g_sMACH.ERR.dwCat3_Error.11 := FALSE;
g_sMACH.ERR.dwCat3_Error.12 := FALSE;
g_sMACH.ERR.dwCat3_Error.13 := FALSE;
g_sMACH.ERR.dwCat3_Error.14 := FALSE;
g_sMACH.ERR.dwCat3_Error.15 := FALSE;

(* --------------------------------------------------------------------------
 * Assign errors of category 4 (Kill automatic sequence)
 * -------------------------------------------------------------------------- *)
g_sMACH.ERR.dwCat4_Error_a.0	:= NOT g_bDI_ES_DirectOK;
g_sMACH.ERR.dwCat4_Error_a.1	:= g_sMACH.ERR.bPressure;
g_sMACH.ERR.dwCat4_Error_a.2	:= FALSE;
g_sMACH.ERR.dwCat4_Error_a.3	:= FALSE;	//g_sMACH.ERR.bErrorArrayTooSmallDia1
									//	OR	g_sMACH.ERR.bErrorArrayTooSmallDia2
									//	OR	g_sMACH.ERR.bErrorArrayTooSmallHor
									//	OR	g_sMACH.ERR.bErrorArrayTooSmallVer;
g_sMACH.ERR.dwCat4_Error_a.4	:= FALSE;	//g_sMACH.ERR.bErrorPosDia1
									//	OR	g_sMACH.ERR.bErrorPosDia2
									//	OR	g_sMACH.ERR.bErrorPosHor
									//	OR	g_sMACH.ERR.bErrorPosVer;
g_sMACH.ERR.dwCat4_Error_a.5	:= g_sMACH.ERR.bUltrasonic1;
g_sMACH.ERR.dwCat4_Error_a.6	:= NOT g_bDI_CircuitBreaker_i700;
g_sMACH.ERR.dwCat4_Error_a.7	:= NOT g_bDI_CircuitBreaker_Ultrasonic;
g_sMACH.ERR.dwCat4_Error_a.8 := g_sMACH.ERR.bServoPowerNOK;
g_sMACH.ERR.dwCat4_Error_a.9 := (g_uStatus_X_Axis.xDriveError OR g_uStatus_X_Axis.xAxisError OR g_uStatus_X_Axis.bLuMessage) AND g_bDI_CircuitBreaker_i700;
g_sMACH.ERR.dwCat4_Error_a.10 := (g_uStatus_Y_Axis.xDriveError OR g_uStatus_Y_Axis.xAxisError OR g_uStatus_Y_Axis.bLuMessage) AND g_bDI_CircuitBreaker_i700;
g_sMACH.ERR.dwCat4_Error_a.11 := (g_uStatus_Z_Axis.xDriveError OR g_uStatus_Z_Axis.xAxisError OR g_uStatus_Z_Axis.bLuMessage) AND g_bDI_CircuitBreaker_i700;
g_sMACH.ERR.dwCat4_Error_a.12 := (g_uStatus_R_Axis.xDriveError OR g_uStatus_R_Axis.xAxisError OR g_uStatus_R_Axis.bLuMessage) AND g_bDI_CircuitBreaker_i700;
g_sMACH.ERR.dwCat4_Error_a.13 := (g_uStatus_Front_Axis.xDriveError OR g_uStatus_Front_Axis.xAxisError OR g_uStatus_Front_Axis.bLuMessage) AND g_bDI_CircuitBreaker_i700;
g_sMACH.ERR.dwCat4_Error_a.14 := (g_uStatus_Rear_Axis.xDriveError OR g_uStatus_Rear_Axis.xAxisError OR g_uStatus_Rear_Axis.bLuMessage) AND g_bDI_CircuitBreaker_i700;
g_sMACH.ERR.dwCat4_Error_a.15 := g_sMACH.ERR.ModusRV_AccDeccZ;
g_sMACH.ERR.dwCat4_Error_a.16 := g_sMACH.ERR.ModusRV_SpeedZToHigh;
g_sMACH.ERR.dwCat4_Error_a.17 := g_sMACH.ERR.ModusRV_TargetPosInSWLimits;
g_sMACH.ERR.dwCat4_Error_a.18 := NOT Front_Axis.xCommunicationOK;
g_sMACH.ERR.dwCat4_Error_a.19 := NOT Rear_Axis.xCommunicationOK;
g_sMACH.ERR.dwCat4_Error_a.20 := NOT Z_Axis.xCommunicationOK;
g_sMACH.ERR.dwCat4_Error_a.21 := NOT R_Axis.xCommunicationOK;
g_sMACH.ERR.dwCat4_Error_a.22 :=g_sMACH.ERR.bErrorComIOStation;
g_sMACH.ERR.dwCat4_Error_a.23 := g_sMACH.ERR.bPieceTooLarge;
g_sMACH.ERR.dwCat4_Error_a.24 := g_sMACH.ERR.bLanguageValueInvalid;
g_sMACH.ERR.dwCat4_Error_a.25 := FALSE;//g_sMACH.sAxisR.bDetectionError;
g_sMACH.ERR.dwCat4_Error_a.26 := FALSE;//g_sMACH.sAxisR.bFollowingError;
g_sMACH.ERR.dwCat4_Error_a.27 := g_sMACH.ERR.bTrayTooSmall;
g_sMACH.ERR.dwCat4_Error_a.28 := g_sMACH.ERR.bR_AxisPositionError;
g_sMACH.ERR.dwCat4_Error_a.29 := g_sMACH.ERR.bAxisFrontNotSet;
g_sMACH.ERR.dwCat4_Error_a.30 := g_sMACH.ERR.bAxisRearNotSet;
g_sMACH.ERR.dwCat4_Error_a.31 := g_sMACH.ERR.bAxisRNotSet;

g_sMACH.ERR.dwCat4_Error_b.00 := g_sMACH.ERR.bWrongTable;
g_sMACH.ERR.dwCat4_Error_b.01 := 	g_sMACH.ERR.bZStrokeKnifeToBottomRound
								OR	g_sMACH.ERR.bZStrokeKnifeToBottomSlab
								OR	g_sMACH.ERR.bZStrokeKnifeToBottomTraySmall
								OR	g_sMACH.ERR.bZStrokeKnifeToBottomTrayLarge
								OR	g_sMACH.ERR.bZStrokeKnifeToBottomTrayDouble;
g_sMACH.ERR.dwCat4_Error_b.02 := 	g_sMACH.ERR.bRoundCakeTooLarge;
g_sMACH.ERR.dwCat4_Error_b.03 := 	g_sMACH.ERR.bSlabTooSmall;
g_sMACH.ERR.dwCat4_Error_b.04 := 	g_sMACH.ERR.bXYNotEnabled;
g_sMACH.ERR.dwCat4_Error_b.05 := 	g_sMACH.ERR.bZNotEnabled;
g_sMACH.ERR.dwCat4_Error_b.06 := 	g_sMACH.ERR.bRNotEnabled;
g_sMACH.ERR.dwCat4_Error_b.07 := 	g_sMACH.ERR.bCleaningContainerZeroPos;
g_sMACH.ERR.dwCat4_Error_b.08 := 	g_sMACH.ERR.bCleaningContainerEndPos;
g_sMACH.ERR.dwCat4_Error_b.09 := 	g_sMACH.ERR.bCleaningContainerEndZero;
g_sMACH.ERR.dwCat4_Error_b.10 := 	g_sMACH.ERR.bCleaningContainerNotSafeToMove;
g_sMACH.ERR.dwCat4_Error_b.11 := 	g_sMACH.ERR.bTableMovementNotAllowed;
g_sMACH.ERR.dwCat4_Error_b.12 := 	g_sMACH.ERR.bRAxisMovementNotAllowed;
g_sMACH.ERR.dwCat4_Error_b.13 := 	g_sMACH.ERR.bZAxisMovementNotAllowed;
g_sMACH.ERR.dwCat4_Error_b.14 := 	g_sMACH.ERR.bZHomeSensorTimeout;
g_sMACH.ERR.dwCat4_Error_b.15 := 	g_sMACH.ERR.bCrashDetectFault;
g_sMACH.ERR.dwCat4_Error_b.16 :=	g_sMACH.ERR.bStackIsFull;							//Tried to push item to stack but stack was full
g_sMACH.ERR.dwCat4_Error_b.17 :=	g_sMACH.ERR.bStackIsEmpty;                          //Tried to pop item from stack but stack was empty
g_sMACH.ERR.dwCat4_Error_b.18 :=	g_sMACH.ERR.bMarginsInOvershootCorrectionInvalid;   //Occurs when marginMax is smaller than marginMin
g_sMACH.ERR.dwCat4_Error_b.19 :=	g_sMACH.ERR.bKnifeSettingsIncorrect;                //Occurs when the knifecenter is bigger than the knife length
g_sMACH.ERR.dwCat4_Error_b.20 :=	g_sMACH.ERR.bIntersectionNotFound;                  //Overshoot detected a collision, but the intersection coulnt be determained
g_sMACH.ERR.dwCat4_Error_b.21 :=	g_sMACH.ERR.bOvershootCorrectionImpossible AND NOT g_HMI_MCH_Parameters.bSkipImpossiblePositions;         //Overshoot coulnt be corrected.
g_sMACH.ERR.dwCat4_Error_b.22 :=	g_sMACH.ERR.bOldOvershootCorrectionDiffers;         //The old overshoot correction still changed the target after the new correction was executed.
g_sMACH.ERR.dwCat4_Error_b.23 :=	g_sMACH.ERR.bIndexOutOfBoundsWhileCopyingCuts;      //Index out of boundaries of array while copying cuts
g_sMACH.ERR.dwCat4_Error_b.24 :=	g_sMACH.ERR.bRoundProductsOverlap;                  //Occurs when round products are to close to eachother, space between them is negative.
g_sMACH.ERR.dwCat4_Error_b.25 :=	g_sMACH.ERR.bCalcVerError;                          //Calc_Ver returned an error.
g_sMACH.ERR.dwCat4_Error_b.26 :=	g_sMACH.ERR.bCalcHorError;                          //Calc_Hor returned an error.
g_sMACH.ERR.dwCat4_Error_b.27 :=	g_sMACH.ERR.bCalcDia1Error;                         //Calc_Dia1 returned an error.
g_sMACH.ERR.dwCat4_Error_b.28 :=	g_sMACH.ERR.bCalcDia2Error;                         //Calc_Dia2 returned an error.
g_sMACH.ERR.dwCat4_Error_b.29 :=	g_sMACH.ERR.bXYA_K_WasNotZero;					    //Thrown when the "k" parameter of a XYA-target wasn't zero, the overshoot correction doent's support this yet.

(* --------------------------------------------------------------------------
 * Error category detection.
 * Only one error category can be active. Errors of higher category take
 * precedence over lower categories
 * -------------------------------------------------------------------------- *)

(* Collect Errors of Category 4 *)
g_sMACH.ERH.bErrorCategory4 :=		g_sMACH.ERR.dwCat4_Error_a <>0
										OR	g_sMACH.ERR.dwCat4_Error_b <>0
										OR	g_sMACH.ERR.dwCat4_Error_c <>0;

 (* Collect Errors of Category 3 *)
g_sMACH.ERH.bErrorCategory3 :=	NOT	g_sMACH.ERH.bErrorCategory4
										AND	g_sMACH.ERR.dwCat3_Error <> 0;

 (* Collect Errors of Category 2 *)
g_sMACH.ERH.bErrorCategory2 :=	NOT		g_sMACH.ERH.bErrorCategory4
										AND NOT	g_sMACH.ERH.bErrorCategory3
										AND		g_sMACH.ERR.dwCat2_Error <>0;

 (* Collect Errors of Category 1 *)
g_sMACH.ERH.bErrorCategory1 :=	NOT		g_sMACH.ERH.bErrorCategory4
										AND NOT	g_sMACH.ERH.bErrorCategory3
										AND NOT	g_sMACH.ERH.bErrorCategory2
										AND		g_sMACH.ERR.dwCat1_Error <> 0;

(* Error request reset handling.
 * --------------------------------------------------------------------------
 * If an error of category 2,3 or 4 occures, the buzzer will sound. It
 * will stop if either a) a maximum time is exceeded (only error category 1) or
 *							b) the HMI.bResetError signal is raised
 * The actual reset error signal (MCL.bResetError) will not be generated as
 * long as the buzzer sounds. In practice this means: the first ResetError
 * keypress will stop the buzzer, the second keypress will reset the error.
 * -------------------------------------------------------------------------- *)

(* Generate oneshots on raising edges of the error categories *)
g_sMACH.ERH.RT_ErrorCategory1(CLK := g_sMACH.ERH.bErrorCategory1);
g_sMACH.ERH.RT_ErrorCategory2(CLK := g_sMACH.ERH.bErrorCategory2);
g_sMACH.ERH.RT_ErrorCategory3(CLK := g_sMACH.ERH.bErrorCategory3);
g_sMACH.ERH.RT_ErrorCategory4(CLK := g_sMACH.ERH.bErrorCategory4);

(* Oneshot on the raising edge of MACH.MCL.bResetErrorPulse *)
g_sMACH.ERH.RT_ResetErrorERH(CLK:=g_HMI_MachCommand.CMD.bResetErrorPulse);

(* Error in category 2,3 or 4 active *)
g_sMACH.ERH.bError234Active :=		  g_sMACH.ERH.bErrorCategory2
										OR	  g_sMACH.ERH.bErrorCategory3
										OR	  g_sMACH.ERH.bErrorCategory4;

(* ----------------------------- *)
(* Handle Buzzer					  *)
(* ----------------------------- *)
(*Blinker for beeping*)
Blinker(Enable:=g_sMACH.ERH.bSoundSignalOn,Timelow:= T#500ms, Timehigh:=T#500ms);
g_bDQ_Buzzer := g_sMACH.ERH.bSoundSignalOn AND Blinker.OUT;

(* Buzzer switch on *)
IF		 (			g_sMACH.ERH.RT_ErrorCategory1.Q
		 AND NOT g_sMACH.ERH.bErrorCategory2
		 AND NOT g_sMACH.ERH.bErrorCategory3
		 AND NOT g_sMACH.ERH.bErrorCategory4
		)
	OR (		  	g_sMACH.ERH.RT_ErrorCategory2.Q
		 AND NOT g_sMACH.ERH.bErrorCategory3
		 AND NOT g_sMACH.ERH.bErrorCategory4
		)
	OR (		  g_sMACH.ERH.RT_ErrorCategory3.Q
		 AND NOT g_sMACH.ERH.bErrorCategory4
		)
	OR (		  g_sMACH.ERH.RT_ErrorCategory4.Q
		)
THEN
	IF		bSkipFirstTrigger
	THEN
			bSkipFirstTrigger := FALSE;
	ELSE
			IF NOT (g_sMACH.ERR.bPressStartToCut AND g_HMI_MachCommand.bScanMode)
			THEN
				g_sMACH.ERH.bSoundSignalOn := TRUE;
			END_IF
	END_IF
END_IF

(* Buzzer timer *)
tBuzzerTimerErr1(IN:= (g_sMACH.ERH.bSoundSignalOn AND NOT g_sMACH.ERH.bError234Active), PT:= T#1s);
tBuzzerTimerErr234(IN:= (g_sMACH.ERH.bSoundSignalOn AND g_sMACH.ERH.bError234Active), PT:= T#3s);

(* Buzzer switch off *)
IF			g_sMACH.ERH.RT_ResetErrorERH.Q
	OR		tBuzzerTimerErr1.Q
	OR		tBuzzerTimerErr234.Q
THEN
			  g_sMACH.ERH.bSoundSignalOn := FALSE;
END_IF

END_PROGRAM

(* ---- MACH_HMI_Control.pou ---- *)
PROGRAM MACH_HMI_Control
VAR

END_VAR
%LANGUAGE ST
(* Status *)
g_sHMI_Mach_UnitStatus.nActState			:= g_sMACH.MCL.nStepCounter;

IF	g_sMACH.ERH.bError234Active
THEN
	g_sHMI_Mach_UnitStatus.nActState := 10;
END_IF

IF g_sMACH.ERH.bErrorCategory4 THEN
	g_HMI_MachCommand.bTestMode := FALSE;
END_IF

g_sHMI_Mach_UnitStatus.dwCat1_Error					:= g_sMACH.ERR.dwCat1_Error;
g_sHMI_Mach_UnitStatus.dwCat2_Error					:= g_sMACH.ERR.dwCat2_Error;
g_sHMI_Mach_UnitStatus.dwCat3_Error					:= g_sMACH.ERR.dwCat3_Error;
g_sHMI_Mach_UnitStatus.dwCat4_Error_a				:= g_sMACH.ERR.dwCat4_Error_a;
g_sHMI_Mach_UnitStatus.dwCat4_Error_b				:= g_sMACH.ERR.dwCat4_Error_b;
g_sHMI_Mach_UnitStatus.dwCat4_Error_c				:= g_sMACH.ERR.dwCat4_Error_c;

g_sHMI_Mach_UnitStatus.bErrorActiv					:= g_sMACH.ERH.bError234Active;
g_sHMI_Mach_UnitStatus.bWarningActiv				:= g_sMACH.ERH.bErrorCategory1 OR g_sHMI_Mach_UnitStatus.bErrorActiv;
g_sHMI_Mach_UnitStatus.bStateAutomatic 				:= g_sMACH.MCL.nStepCounter = StateAutomatic;
g_sHMI_Mach_UnitStatus.bHomingDone					:= g_bHomingDone;
g_sHMI_Mach_UnitStatus.bProcessBusy					:= g_sMACH.aut.bProcessBusy;
g_sHMI_Mach_UnitStatus.bScanModeBusy				:= g_HMI_MachCommand.bScanMode;
g_sHMI_Mach_UnitStatus.bEmergencyStop				:= NOT g_bDI_ES_DirectOK;
													//OR NOT g_bDI_LightCurtainOK;

g_sHMI_Mach_UnitStatus.dwAGM1_PowerLoss				:= g_dwAGM1_PowerLoss;
g_sHMI_Mach_UnitStatus.rAGM1_Frequency				:= g_rAGM1_Frequency;

(* Positions *)
g_sHMI_Mach_UnitStatus.dnActualPosDrive_X			:= REAL_TO_DINT(g_uStatus_X_Axis.lrActPosition);
g_sHMI_Mach_UnitStatus.dnActualPosDrive_Y			:= REAL_TO_DINT(g_uStatus_Y_Axis.lrActPosition);
g_sHMI_Mach_UnitStatus.dnActualPosDrive_Front		:= REAL_TO_DINT(g_uStatus_Front_Axis.lrActPosition);
g_sHMI_Mach_UnitStatus.dnActualPosDrive_Rear		:= REAL_TO_DINT(g_uStatus_Rear_Axis.lrActPosition);
g_sHMI_Mach_UnitStatus.dnActualPosDrive_Z			:= REAL_TO_DINT(g_uStatus_Z_Axis.lrActPosition);
g_sHMI_Mach_UnitStatus.dnActualPosDrive_R			:=g_uStatus_R_Axis.lrActPosition;

(* Enable Start button *)
g_sHMI_Mach_UnitStatus.wButtonStatus.0				:=	g_sHMI_Mach_UnitStatus.nActState = StateWaitForInit
													OR	g_sHMI_Mach_UnitStatus.nActState = StateWaitForAutomatic
													OR	(g_sHMI_Mach_UnitStatus.nActState = StateAutomatic AND g_sMACH.MCL.bHoldOnRequest);
(* Enable Pause button *)
g_sHMI_Mach_UnitStatus.wButtonStatus.1				:= (g_sHMI_Mach_UnitStatus.nActState = StateAutomatic AND NOT g_sMACH.MCL.bHoldOnRequest);
(* Enable Stop button *)
g_sHMI_Mach_UnitStatus.wButtonStatus.2				:= (g_sHMI_Mach_UnitStatus.nActState = StateAutomatic AND NOT g_sMACH.MCL.bStopEndOfCycle);
(* g_HMI_dwButtonStatus.3	:= gMachConfig.bPneumaticRaxis used for visible SetRef R-axis button *)
(* Enable Cleaning mode button *)
g_sHMI_Mach_UnitStatus.wButtonStatus.4				:=	g_sHMI_Mach_UnitStatus.nActState = StateWaitForRecipe
													OR	g_sHMI_Mach_UnitStatus.nActState = StateWaitForAutomatic;
(* g_HMI_dwButtonStatus.5	used for visible SetRef X-axis button *)

(* Visible van Y richting aantal stukken*)
g_sHMI_MACH_UnitStatus.wButtonStatus.6 	:= g_HMI_RCP_Parameters.nProductType <> Prod_Slab_Rectangle_2x1;

(* Enable Clean once button *)
g_sHMI_Mach_UnitStatus.wButtonStatus.7		:=		g_sHMI_Mach_UnitStatus.nActState = StateWaitForInit
												OR	g_sHMI_Mach_UnitStatus.nActState = StateWaitForAutomatic
												OR	(g_sHMI_Mach_UnitStatus.nActState = StateAutomatic AND g_sMACH.MCL.bHoldOnRequest)
												OR NOT gMachConfig.bCleaningUnit;

(*REDCASE BITS*)
(*Prepare machine*)
g_sHMI_Mach_UnitStatus.wButtonStatus.8		:= g_HMI_MachCommand.bScanMode AND g_sHMI_Mach_UnitStatus.nActState <> StateAutomatic  AND NOT  g_sHMI_Mach_UnitStatus.bScanFinished;;
(*Scan busy*)
g_sHMI_Mach_UnitStatus.wButtonStatus.9		:= g_HMI_MachCommand.bScanMode AND g_sHMI_Mach_UnitStatus.nActState = StateAutomatic AND NOT  g_sHMI_Mach_UnitStatus.bScanFinished;
(*Scan ready but uploading*)
g_sHMI_Mach_UnitStatus.wButtonStatus.10		:= g_HMI_MachCommand.bScanMode AND g_sHMI_Mach_UnitStatus.bScanFinished;
(*Please leave screen*)
g_sHMI_Mach_UnitStatus.wButtonStatus.11		:= NOT g_HMI_MachCommand.bScanMode;

(*Tray product*)
g_sHMI_Mach_UnitStatus.wButtonStatus.12		:= (g_HMI_RCP_Parameters.nProductType = Prod_Tray_Rectangle_1x1
											OR g_HMI_RCP_Parameters.nProductType = Prod_Tray_Rectangle_1x2
											OR g_HMI_RCP_Parameters.nProductType = Prod_Tray_Rectangle_2x1
											OR g_HMI_RCP_Parameters.nProductType = Prod_Tray_Rectangle_1x4)
											AND gMachConfig.bCrashDetection;

(* IO visualisation *)
g_sHMI_Mach_UnitStatus.wInputs_Modul0_1	:= g_byInputs_Module_00 + 256 * g_byInputs_Module_01;
g_sHMI_Mach_UnitStatus.wInputs_Modul2_3	:= g_byInputs_Module_02 + 256 * g_byInputs_Module_03;
g_sHMI_Mach_UnitStatus.wInputs_Modul4_5	:= g_byInputs_Module_04 + 256 * g_byInputs_Module_05;
g_sHMI_Mach_UnitStatus.wOutputs_Modul0_1:= g_byOutputs_Module_00 + 256 * g_byOutputs_Module_01;

(*Reset productCounters*)
IF g_HMI_MachCommand.CMD.bResetDayCounter THEN
	g_sHMI_CountersDay.dnProductCountTotal 			:= 0;
	g_sHMI_CountersDay.dnProductCountTrayLarge		:= 0;
	g_sHMI_CountersDay.dnProductCountTraySmall		:= 0;
	g_sHMI_CountersDay.dnProductCountSlabSquare		:= 0;
	g_sHMI_CountersDay.dnProductCountSlabDiagonal 	:= 0;
	g_sHMI_CountersDay.dnProductCountSlabTriangle 	:= 0;
	g_sHMI_CountersDay.dnProductCountRound 			:= 0;
	g_sHMI_CountersDay.dnProductCountTrayTriple		:= 0;	(* V03.03 *)
END_IF

(* Status light in HMI*)
IF g_sMACH.MCL.nStepCounter >= StateWaitForRecipe THEN
	g_sHMI_Mach_UnitStatus.byStatusInit := 3;
ELSIF g_sMACH.MCL.nStepCounter = StateInit THEN
	g_sHMI_Mach_UnitStatus.byStatusInit := 2;
ELSE
	g_sHMI_Mach_UnitStatus.byStatusInit := 1;
END_IF

(*Triangle choice*)
IF g_HMI_RCP_Parameters.bUseRectanglesForTriangles THEN
	g_sHMI_Mach_UnitStatus.nTrianglesChoice := 2;
ELSIF g_HMI_RCP_Parameters.bUseRectanglesInEight THEN
	g_sHMI_Mach_UnitStatus.nTrianglesChoice := 1;
ELSE
	g_sHMI_Mach_UnitStatus.nTrianglesChoice := 0;
END_IF

(* functions for new Visu *)
g_HMI_RCP_ShowCleaningsettings	:= gMachConfig.bCleaningUnit;
g_HMI_RCP_ShowCrashDetectionSettings := gMachConfig.bCrashDetection;
VisuCutsHandler();
VisuDashboardNotifications();
RecipeChoiceSelector();

IF g_sHMI_Mach_UnitStatus.bEmergencyStop AND NOT(g_HMI_bCloseOverlay) THEN
	g_HMI_bShowOverlay := TRUE;
ELSE
	g_HMI_bShowOverlay := FALSE;
END_IF
IF NOT(g_sHMI_Mach_UnitStatus.bEmergencyStop) THEN
	g_HMI_bCloseOverlay := FALSE;
END_IF

END_PROGRAM

(* ---- MACH_INI_Initialise.pou ---- *)
PROGRAM MACH_INI_Initialise
VAR
	bPulseStepCounter		: BOOL;
	bWait						: BOOL;
	tWatchDogTimer			: TON;
	tStepTimer				: TOF;
END_VAR
%LANGUAGE ST
(*************************************************************************
 *
 * Application name				: Snijmachine
 * Module name					: MACH_INI_Initialise
 * Version number module		: 0.00
 *
 *
 *						Copyright (c) Bakon 2009
 *						Goes, The Netherlands
 *
 *
 * All rights are reserved. Reproduction in whole or in part is prohibited
 * without the written consent of the copyright owner.
 *
 *************************************************************************)

(*************************************************************************
 * HISTORY
 *************************************************************************
 * Update  : 0.00
 * Author  :	 K. Kole
 * Changes :
 *************************************************************************)
(* Force C_NOT_ACTIVE state *)
IF	  NOT g_sMACH.MCL.bActInitialise
THEN
		  g_sMACH.uINI.nStepCounter := C_NOT_ACTIVE;
END_IF

IF		g_sMACH.uINI.nStepCounter <> C_NOT_ACTIVE
THEN
	(* -------------------------------------------------------------------------
	 * Prestep Code
	 * ------------------------------------------------------------------------- *)
				  ;
END_IF;

(* detect change of state *)
bPulseStepCounter	  := g_sMACH.uINI.nStepCounter <> g_sMACH.uINI.nOldStepCounter;
g_sMACH.uINI.nOldStepCounter := g_sMACH.uINI.nStepCounter;

(* Steptimer *)
tStepTimer (IN:= bPulseStepCounter, PT:= REAL_TO_TIME(g_sMACH.uINI.rStepTime));
bWait := tStepTimer.Q;

(* Watchdogtimer *)
tWatchDogTimer (IN:= 	NOT	bPulseStepCounter
						AND		g_sMACH.MCL.bActInitialise
						AND NOT	g_HMI_MachCommand.CMD.bResetErrorPulse
						AND		g_sMACH.uINI.rWatchdogTime <> 0,
					PT:= REAL_TO_TIME(g_sMACH.uINI.rWatchdogTime));
g_sMACH.uINI.bAlmError := tWatchDogTimer.Q;

CASE g_sMACH.uINI.nStepCounter OF
	(* --------------------------------------------------------------------------
	 * S-1  C_NOT_ACTIVE
	 *		OnEntry: Ready  := FALSE
	 *		OnEntry: Busy	:= FALSE
	 *		OnEntry: Reset all non-stored commands
	 * T000 Activate signal
	 * -------------------------------------------------------------------------- *)
	C_NOT_ACTIVE:

		(* On Entry *)
		IF			bPulseStepCounter
		THEN
					g_sMACH.uINI.rWatchdogTime		:= 0;
					g_sMACH.uINI.bInitialiseReady		:= FALSE;
					g_sMACH.uINI.bInitialiseBusy		:= FALSE;
					MACH_SUB_Initialise.I_rX_InfeedPosition		:= g_HMI_MCH_Parameters.rInfeedPosition_X;
					MACH_SUB_Initialise.I_rY_InfeedPosition		:= g_HMI_MCH_Parameters.rInfeedPosition_Y;
					MACH_SUB_Initialise.I_rY_InfeedPrePosition	:= g_HMI_MCH_Parameters.rInfeedPosition_Y + 30;
					g_bSUB_InitStart						:= FALSE;
		END_IF

		(* Continuous actions *)

		(* Transitions *)
		IF		g_sMACH.MCL.bActInitialise
		THEN
				g_sMACH.uINI.nStepCounter			:= C_INITIAL;
		END_IF

	(* --------------------------------------------------------------------------
	 * S000 C_INITIAL
	 *		OnEntry: Ready := FALSE
	 *		OnEntry: Busy  := TRUE
	 *		Start SUB Init
	 * T001 Always
	 * -------------------------------------------------------------------------- *)
	C_INITIAL:

		(* On Entry *)
		IF		bPulseStepCounter
		THEN
				g_sMACH.uINI.rWatchdogTime			:= 0;
				g_sMACH.uINI.bInitialiseReady			:= FALSE;
				g_sMACH.uINI.bInitialiseBusy			:= TRUE;

				g_bSUB_InitStart							:= TRUE;
		END_IF

		(* Continuous actions *)

		(* Transitions *)
		IF		g_bSUB_InitDone
		THEN
				g_bSUB_InitStart					:= FALSE;
				g_sMACH.uINI.nStepCounter		:= C_READY;
		END_IF

	(* --------------------------------------------------------------------------
	 * S998 C_READY
	 *		OnEntry: Ready		:= TRUE
	 *		OnEntry: Busy		 := FALSE
	 *		Always : Activate errorhandler
	 * T000 Never
	 * -------------------------------------------------------------------------- *)
	C_READY:

		(* On Entry *)
		IF			bPulseStepCounter
		THEN
					g_sMACH.uINI.rWatchdogTime	:= 0;
					g_sMACH.uINI.bInitialiseReady		:= TRUE;
					g_sMACH.uINI.bInitialiseBusy		:= FALSE;
		END_IF

		(* Continuous actions *)

		(* Transitions *)
		IF			FALSE
		THEN
					g_sMACH.uINI.nStepCounter				:= C_INITIAL;
		END_IF

(* --------------------------------------------------------------------------
 * Illegal state
 * -------------------------------------------------------------------------- *)
ELSE
	(* Programming error: Illegal state *)
	g_sMACH.uINI.rWatchdogTime := 10;
END_CASE;

IF			g_sMACH.uINI.nStepCounter <> C_NOT_ACTIVE
THEN
	(* -------------------------------------------------------------------------
	 * Poststep Code
	 * ------------------------------------------------------------------------- *)
	;
END_IF

END_PROGRAM

(* ---- MACH_MAN_Manual.pou ---- *)
PROGRAM MACH_MAN_Manual
VAR
	bPulseStepCounter	: BOOL;
	bHoldPointOnReq	: BOOL;
	bHoldPointOnErr3	: BOOL;
END_VAR

%LANGUAGE ST
(*************************************************************************
 *
 * Application name				: Snijmachine
 * Module name					: MACH_MAN_Manual
 * Version number module		: 0.00
 *
 *
 *						Copyright (c) Bakon 2009
 *						Goes, The Netherlands
 *
 *
 * All rights are reserved. Reproduction in whole or in part is prohibited
 * without the written consent of the copyright owner.
 *
 *************************************************************************)

(*************************************************************************
 * HISTORY
 *************************************************************************
 * Update  :
 * Author  :
 * Changes :
 *************************************************************************)

	bHoldPointOnReq		:= FALSE;
	bHoldPointOnErr3		:= FALSE;

	(* Force C_NOT_ACTIVE state *)
	IF	  NOT g_sMACH.MCL.bActManual
	THEN
				  g_sMACH.MAN.nStepCounter := C_NOT_ACTIVE;
	END_IF

	g_sMACH.ERR.bPressStartForManual	:= (g_sMACH.MAN.nStepCounter = C_INITIAL) AND g_bDI_MachineInSafePosition;

	IF			g_sMACH.MAN.nStepCounter <> C_NOT_ACTIVE
	THEN
	(* -------------------------------------------------------------------------
	 * Prestep Code
	 * ------------------------------------------------------------------------- *)
				;
	END_IF

	(* detect change of state *)
	bPulseStepCounter					:= g_sMACH.MAN.nStepCounter <> g_sMACH.MAN.nOldStepCounter;
	g_sMACH.MAN.nOldStepCounter	:= g_sMACH.MAN.nStepCounter;

	(* Steptimer *)

	(* Watchdogtimer *)

	CASE g_sMACH.MAN.nStepCounter OF
	(* --------------------------------------------------------------------------
	 *  S-1  C_NOT_ACTIVE
	 *		 OnEntry: Ready  := FALSE
	 *		 OnEntry: Busy	:= FALSE
	 *		 OnEntry: InHold := FALSE
	 *		 OnEntry: Reset all non-stored commands
	 *  T000 Activate signal
	 * -------------------------------------------------------------------------- *)
	C_NOT_ACTIVE:

		(* On Entry *)
		IF			bPulseStepCounter
		THEN
					g_sMACH.MAN.bManualReady					:= FALSE;
					g_sMACH.MAN.bManualBusy					:= FALSE;
					g_sMACH.MAN.bManualHold						:= FALSE;
					(*g_uControl_X_Axis.bStartManualMode			:= FALSE;
					g_uControl_Y_Axis.bStartManualMode			:= FALSE;
					g_uControl_Front_Axis.bStartManualMode		:= FALSE;
					g_uControl_Rear_Axis.bStartManualMode		:= FALSE;
					g_uControl_Front_Axis.bAutomatic				:= FALSE;
					g_uControl_Rear_Axis.bStartManualMode		:= FALSE;
					g_uControl_Rear_Axis.bAutomatic				:= FALSE;
					g_uControl_Z_Axis.bStartManualMode			:= FALSE;
					g_uControl_R_Axis.bStartManualMode			:= FALSE;*)
					g_uControl_X_Axis.bManualJogPos				:= FALSE;
					g_uControl_X_Axis.bManualJogNeg				:= FALSE;
					g_uControl_Y_Axis.bManualJogPos				:= FALSE;
					g_uControl_Y_Axis.bManualJogNeg				:= FALSE;
					g_uControl_Front_Axis.bManualJogPos			:= FALSE;
					g_uControl_Front_Axis.bManualJogNeg			:= FALSE;
					g_uControl_Rear_Axis.bManualJogPos			:= FALSE;
					g_uControl_Rear_Axis.bManualJogNeg			:= FALSE;
					g_uControl_Z_Axis.bManualJogPos				:= FALSE;
					g_uControl_Z_Axis.bManualJogNeg				:= FALSE;
					g_uControl_R_Axis.bManualJogPos				:= FALSE;
					g_uControl_R_Axis.bManualJogNeg				:= FALSE;
					g_bCMD_US_Test1								:= FALSE;
					g_HMI_MachCommand.bSetOffsetR				:= FALSE;
					g_HMI_MachCommand.bSetOffsetFront			:= FALSE;
					g_HMI_MachCommand.bSetOffsetRear			:= FALSE;
					g_sMACH.sCleaningContainerControl.bManual	:= FALSE;
					g_sMACH.sCleaningContainerControl.bManualNeg	:= FALSE;
					g_sMACH.sCleaningContainerControl.bManualPos	:= FALSE;
					g_bDQ_CleaningWaterValve		:= 		FALSE;
		END_IF

		(* Continuous actions *)
		(* Reset manual functions active/selectable bits *)

		(* Transitions *)
		IF			g_sMACH.MCL.bActManual
		THEN
					g_sMACH.MAN.nStepCounter			:= C_INITIAL;
		END_IF

	(*--------------------------------------------------------------------------
	 *  S000 C_INITIAL
	 *		 OnEntry: Ready := FALSE
	 		Wait for start button
	 *  T001 Startbutton pressed
	 * -------------------------------------------------------------------------- *)
	C_INITIAL:

		(* On Entry *)
		IF			bPulseStepCounter
		THEN
					g_sMACH.MAN.bManualReady  := FALSE;
		END_IF

		(* Continuous actions *)

		(* Transitions *)
		IF		g_sMACH.MCL.bStopEndOfCycle
		THEN
				g_sMACH.MAN.nStepCounter			:= C_READY;
		ELSIF				g_bDI_StartButton
				OR NOT	g_bDI_MachineInSafePosition
		THEN
				g_sMACH.MAN.nStepCounter			:= 001;
		END_IF

	(*--------------------------------------------------------------------------
	 *  S001 Enable drives
	 *  T002 Status Manual mode of the drives
	 * -------------------------------------------------------------------------- *)
	001:

		(* On Entry *)
		IF			bPulseStepCounter
		THEN
					g_uControl_X_Axis.bEnableDrive	:= TRUE;
					g_uControl_Y_Axis.bEnableDrive	:= TRUE;
					g_uControl_Front_Axis.bEnableDrive	:= TRUE;
					g_uControl_Rear_Axis.bEnableDrive	:= TRUE;
					g_uControl_Z_Axis.bEnableDrive	:= TRUE;
					g_uControl_R_Axis.bEnableDrive	:= TRUE;
					g_sMACH.sCleaningContainerControl.bManual	:= TRUE;

					g_uControl_X_Axis.lrDeceleration	:=X_Axis.scPar.MaxAcceleration;	//Was fSWMaxDeceleration in old motion
					g_uControl_Y_Axis.lrDeceleration	:=Y_Axis.scPar.MaxAcceleration;	//Was fSWMaxDeceleration in old motion
					g_uControl_Front_Axis.lrDeceleration	:=Front_Axis.scPar.MaxAcceleration;	//Was fSWMaxDeceleration in old motion
					g_uControl_Rear_Axis.lrDeceleration	:=Rear_Axis.scPar.MaxAcceleration;	//Was fSWMaxDeceleration in old motion
					g_uControl_Z_Axis.lrDeceleration	:=Z_Axis.scPar.MaxAcceleration;	//Was fSWMaxDeceleration in old motion
					g_uControl_R_Axis.lrDeceleration	:=R_Axis.scPar.MaxAcceleration;	//Was fSWMaxDeceleration in old motion

					(*g_uControl_X_Axis.bStartManualMode	:= TRUE;
					g_uControl_Y_Axis.bStartManualMode	:= TRUE;
					g_uControl_Front_Axis.bAutomatic		:= TRUE;
					g_uControl_Rear_Axis.bAutomatic		:= TRUE;
					g_uControl_Z_Axis.bStartManualMode	:= TRUE;
					g_uControl_R_Axis.bStartManualMode	:= TRUE;*)

		END_IF

		(* Continuous actions *)
		Calc_BottomPos();

		(* Transitions *)
		IF		g_sMACH.MCL.bStopEndOfCycle
		THEN
				g_sMACH.MAN.nStepCounter			:= C_READY;
		ELSIF		g_uStatus_X_Axis.bDriveEnabled
			AND	g_uStatus_Y_Axis.bDriveEnabled
			AND	g_uStatus_Front_Axis.bDriveEnabled
			AND	g_uStatus_Rear_Axis.bDriveEnabled
			AND	g_uStatus_Z_Axis.bDriveEnabled
			AND	g_uStatus_R_Axis.bDriveEnabled
		THEN
					  g_sMACH.MAN.nStepCounter			:= 002;
		END_IF

	(* --------------------------------------------------------------------------
	 *  S002 All movements
	 *  T998 Never
	 * -------------------------------------------------------------------------- *)
	002:

		(* On Entry *)
		IF			bPulseStepCounter
		THEN
			;
		END_IF

		(* Continuous actions *)
		g_uControl_X_Axis.bManualJogPos			:= g_HMI_MachCommand.bMan_XaxisPos;
		g_uControl_X_Axis.bManualJogNeg			:= g_HMI_MachCommand.bMan_XaxisNeg;
		g_uControl_Y_Axis.bManualJogPos			:= g_HMI_MachCommand.bMan_YaxisPos;
		g_uControl_Y_Axis.bManualJogNeg			:= g_HMI_MachCommand.bMan_YaxisNeg;
		g_uControl_Front_Axis.bManualJogPos		:= g_HMI_MachCommand.bMan_FrontaxisPos;
		g_uControl_Front_Axis.bManualJogNeg		:= g_HMI_MachCommand.bMan_FrontaxisNeg;
		g_uControl_Rear_Axis.bManualJogPos		:= g_HMI_MachCommand.bMan_RearaxisPos;
		g_uControl_Rear_Axis.bManualJogNeg		:= g_HMI_MachCommand.bMan_RearaxisNeg;
		g_uControl_Z_Axis.bManualJogPos			:= g_HMI_MachCommand.bMan_ZaxisPos;
		g_uControl_Z_Axis.bManualJogNeg			:= g_HMI_MachCommand.bMan_ZaxisNeg;
		g_uControl_R_Axis.bManualJogPos			:= g_HMI_MachCommand.bMan_RaxisPos;
		g_uControl_R_Axis.bManualJogNeg			:= g_HMI_MachCommand.bMan_RaxisNeg;
		g_bCMD_US_Test1							:= g_HMI_MachCommand.bTestUltrasonic1;

		(* Cleaning container *)
		g_sMACH.sCleaningContainerControl.bManualPos		:= g_HMI_MachCommand.bMan_CleaningContPos;
		g_sMACH.sCleaningContainerControl.bManualNeg		:= g_HMI_MachCommand.bMan_CleaningContNeg;

		(* Water valve *)
		g_bDQ_CleaningWaterValve		:= g_HMI_MachCommand.bMan_CleaningWaterPos;

		(* Transitions *)
		IF			g_sMACH.MCL.bStopEndOfCycle
		THEN
					g_sMACH.MAN.nStepCounter			:= C_READY;
		END_IF

	(* --------------------------------------------------------------------------
	 *  S998 C_READY
	 *  T000 Always
	 * -------------------------------------------------------------------------- *)
	C_READY:

		(* On Entry *)
		IF			bPulseStepCounter
		THEN
					g_sMACH.MAN.rWatchdogTime	  := 0;
		END_IF

		(* Continuous actions *)
		g_sMACH.MAN.bManualReady	:= TRUE;

		(* Transitions *)
		IF			TRUE
		THEN
					g_sMACH.MAN.nStepCounter			:= C_INITIAL;
		END_IF

	(* --------------------------------------------------------------------------
	 * Illegal state
	 * -------------------------------------------------------------------------- *)
	ELSE
		(* Programming error: Illegal state *)
		g_sMACH.MAN.rWatchdogTime := 10;
	END_CASE;

	IF		 g_sMACH.MAN.nStepCounter <> C_NOT_ACTIVE
	THEN
	(* -------------------------------------------------------------------------
	 * Poststep Code
	 * ------------------------------------------------------------------------- *)

				g_sMACH.MAN.bManualHold := FALSE;

				g_sMACH.MAN.bManualBusy :=			g_sMACH.MCL.bActManual
											  AND NOT g_sMACH.MAN.bManualHold;

	END_IF

END_PROGRAM
